// TwinCAT 3 PLC project mobject_graph_vision_pack
// Title: mobject-graph-vision-pack
// Company: mobject
// Author: mobject dev team
// ProjectVersion: 0.11.0
// ProgramVersion: 3.1.4026.25
// libraries:
//   mobject-core,0.10.0,mobject
//   mobject-graph,0.18.0,mobject
//   mobject-graph-plc-pack,0.19.0,mobject
//   Tc2_Standard, * (Beckhoff Automation GmbH)
//   Tc2_System, * (Beckhoff Automation GmbH)
//   Tc2_Utilities, * (Beckhoff Automation GmbH)
//   Tc3_Module, * (Beckhoff Automation GmbH)
//   Tc3_Vision, 5.10.2.0 (Beckhoff Automation GmbH)
// project tree:
//   Datatypes/Aliases/ _GVCP_REGISTER_ADDRESS.TcPOU, _TcVnMatrix2x3_LREAL.TcPOU, _TcVnArray4_Point2_REAL.TcPOU (not stored), _TcVnArray4_LREAL.TcPOU (not stored), _TcVnArray33_UDINT.TcPOU (not stored), _TcVnArray10_ITcVnImage.TcPOU (not stored), _TcVnArray3_Point2_REAL.TcPOU (not stored), _TcVnArray7_LREAL.TcPOU, _TcVnArray8_LREAL.TcPOU, _TcVnMatrix3x3_LREAL.TcPOU (not stored), _TcVnPoint.TcPOU (not stored), _TcVnPoint2_LREAL.TcPOU (not stored), _TcVnPoint3_REAL.TcPOU, _TcVnPoint3_LREAL.TcPOU, _TcVnPoint2_REAL.TcPOU (not stored), _TcVnRectangle.TcPOU (not stored), _TcVnVector2_DINT.TcPOU, _TcVnPoint2_DINT.TcPOU (not stored), _ALIASTYP.TcPOU (not stored) (excluded from build), _TcVnVector2_INT.TcPOU (not stored), _TcVnVector3_SINT.TcPOU (not stored), _TcVnVector3_INT.TcPOU, _TcVnVector2_SINT.TcPOU (not stored), _TcVnVector2_LREAL.TcPOU (not stored), _TcVnVector2_UINT.TcPOU (not stored), _TcVnVector2_USINT.TcPOU, _TcVnVector3_UINT.TcPOU, _TcVnVector3_USINT.TcPOU (not stored), _TcVnVector4_INT.TcPOU (not stored), _TcVnVector4_REAL.TcPOU, _TcVnVector4_SINT.TcPOU (not stored), _TcVnVector4_LREAL.TcPOU (not stored), _TcVnVector3_REAL.TcPOU, _TcVnVector3_LREAL.TcPOU (not stored), _TcVnVector2_REAL.TcPOU (not stored), _TcVnVector4_DINT.TcPOU, _TcVnVector4_UINT.TcPOU, _TcVnVector4_USINT.TcPOU, _GVCP_REGISTER_VALUE.TcPOU
//   Datatypes/Arrays/ _Array0to1OfARRAYTYP.TcPOU (not stored) (excluded from build), _Array0to1OfDINT.TcPOU (not stored), _Array0to1OfINT.TcPOU, _Array0to1OfLREAL.TcPOU (not stored), _Array0to1OfREAL.TcPOU (not stored), _Array0to1OfSINT.TcPOU, _Array0to1OfUINT.TcPOU (not stored), _Array0to1OfUSINT.TcPOU, _Array0to1_0to2OfLREAL.TcPOU, _Array0to2_0to2OfLREAL.TcPOU (not stored), _Array0to2OfINT.TcPOU (not stored), _Array0to2OfLREAL.TcPOU (not stored), _Array0to2OfREAL.TcPOU, _Array0to2OfSINT.TcPOU, _Array0to2OfTcVnPoint2_REAL.TcPOU (not stored), _Array0to2OfUINT.TcPOU (not stored), _Array0to2OfUSINT.TcPOU (not stored), _Array0to32OfUDINT.TcPOU (not stored), _Array0to3OfDINT.TcPOU (not stored), _Array0to3OfINT.TcPOU, _Array0to3OfLREAL.TcPOU, _Array0to3OfREAL.TcPOU, _Array0to3OfSINT.TcPOU (not stored), _Array0to3OfTcVnPoint2_REAL.TcPOU, _Array0to3OfUINT.TcPOU, _Array0to3OfUSINT.TcPOU (not stored), _Array0to6OfLREAL.TcPOU (not stored), _Array0to7OfLREAL.TcPOU, _Array0to9OfITcVnImage.TcPOU
//   Datatypes/Enums/ _ETcVn2dCodeSearchStrategy.TcPOU (not stored), _ETcVnCodeType.TcPOU, _ETcVnMatchTemplateWalshOptions.TcPOU, _ETcVnCodeDetectionModel.TcPOU, _ETcVnAdaptiveThresholdMethod.TcPOU (not stored), _ETcVnBarcodeSearchDirection.TcPOU (not stored), _ETcVnBarcodeType.TcPOU (not stored), _ETcVnBlobCombination.TcPOU (not stored), _ETcVnBorderInterpolationMethod.TcPOU (not stored), _ETcVnBoostClassifierType.TcPOU, _ETcVnCalibrationPattern.TcPOU (not stored), _ETcVnCalibrationPatternOrigin.TcPOU, _ETcVnCameraState.TcPOU, _ETcVnClusteringAlgorithm.TcPOU, _ETcVnColorMap.TcPOU (not stored), _ETcVnColorMapSize.TcPOU, _ETcVnColorSpaceTransform.TcPOU, _ETcVnColorTrainingMethod.TcPOU, _ETcVnConnectedComponentsAlgorithm.TcPOU, _ETcVnContainerExportFormat.TcPOU (not stored), _ETcVnContourApproximationMethod.TcPOU (not stored), _ETcVnContourRetrievalMode.TcPOU (not stored), _ETcVnContoursMatchComparisonMethod.TcPOU (not stored), _ETcVnDataMatrixOptions.TcPOU, _ETcVnFindTemplateWalshOptions.TcPOU, _ETcVnReduceType.TcPOU, _ETcVnDiffusivityTypeKAZE.TcPOU (not stored), _ETcVnDistanceTransformationLabel.TcPOU, _ETcVnDistanceTransformationMask.TcPOU, _ETcVnDistanceType.TcPOU, _ETcVnDrawMatchesFlags.TcPOU, _ETcVnDrawShape.TcPOU, _ETcVnEdgeDetectionAlgorithm.TcPOU (not stored), _ETcVnEdgeDirection.TcPOU, _ETcVnElementType.TcPOU (not stored), _ETcVnEstimationAlgorithm.TcPOU (not stored), _ETcVnExtremePointDirection.TcPOU, _ETcVnFeatureDescriptorTypeAKAZE.TcPOU, _ETcVnFeatureScalingType.TcPOU, _ETcVnFeatureScoreTypeORB.TcPOU (not stored), _ETcVnFilterDirection.TcPOU (not stored), _ETcVnFlipAxis.TcPOU, _ETcVnDataLayout.TcPOU, _ETcVnFontType.TcPOU, _ETcVnHoughMethod.TcPOU (not stored), _ETcVnInitializableFunction.TcPOU, _ETcVnInterpolationType.TcPOU (not stored), _ETcVnKeypointDetectionTypeAGAST.TcPOU, _ETcVnKeypointDetectionTypeFAST.TcPOU (not stored), _ETcVnKnn.TcPOU (not stored), _ETcVnLineType.TcPOU, _ETcVnMorphologicalOperator.TcPOU, _ETcVnNbc.TcPOU (not stored), _ETcVnNormalizationType.TcPOU (not stored), _ETcVnOcrModelType.TcPOU, _ETcVnCircularityCalculationMethod.TcPOU, _ETcVnLayerNameType.TcPOU, _ETcVnTimestamp.TcPOU, _ETcVnOcrOptions.TcPOU, _ETcVnOrientationMethod.TcPOU (not stored), _ETcVnPaddingMode.TcPOU (not stored), _ETcVnPixelConnectivity.TcPOU, _ETcVnPixelEncoding.TcPOU (not stored), _ETcVnPixelPackMode.TcPOU, _ETcVnPrototypeClusterer.TcPOU (not stored), _ETcVnRectangleIntersection.TcPOU, _ETcVnRotationAngle.TcPOU, _ETcVnRTrees.TcPOU (not stored), _ETcVnSignedNormalization.TcPOU (not stored), _ETcVnSolvePnPMethod.TcPOU (not stored), _ETcVnSta.TcPOU (not stored), _ETcVnStructuringElementShape.TcPOU, _ETcVnSvm.TcPOU (not stored), _ETcVnSvmKernelType.TcPOU (not stored), _ETcVnSvmSgdClassifierMarginType.TcPOU, _ETcVnSvmSgdClassifierType.TcPOU (not stored), _ETcVnTemplateMatchMethod.TcPOU (not stored), _ETcVnThresholdType.TcPOU, _ETcVnVectorCompareMethod.TcPOU (not stored), _ETcVnWorldCoordinateSystem.TcPOU (not stored), _ETcWatchdogAccumulationType.TcPOU (not stored), _GEV_CAMERA_STATE.TcPOU, _ETcVnComparisonOperator.TcPOU, _ETcVnDetectBarcodesWalshOptions.TcPOU, _ETcVnDetectPatternPointsOptions.TcPOU, _ETcVnDotCodeOptions.TcPOU, _ETcVnEdgeSelection.TcPOU, _ETcVnFindRoisMethod.TcPOU, _ETcVnJpegSampling.TcPOU, _ETcVnMergeRegionsOptions.TcPOU, _ETcVnPolarizedImageInterpolation.TcPOU, _ETcVnSalientFeaturesMethod.TcPOU
//   Datatypes/Interfaces/Containers/ITcVnContainer/ I_InterfaceDatatype_ITcVnContainer.TcIO (not stored), _ITcVnContainer.TcPOU (not stored)
//   Datatypes/Interfaces/Containers/Iterators/ITcVnBidirectionalIterator/ I_InterfaceDatatype_ITcVnBidirectionalIterator.TcIO (not stored), _ITcVnBidirectionalIterator.TcPOU (not stored)
//   Datatypes/Interfaces/Images/ITcVnImage/ I_InterfaceDatatype_ITcVnImage.TcIO (not stored), _ITcVnImage.TcPOU (not stored)
//   Datatypes/Interfaces/Images/ITcVnDisplayableImage/ I_InterfaceDatatype_ITcVnDisplayableImage.TcIO (not stored), _ITcVnDisplayableImage.TcPOU (not stored)
//   Datatypes/Structs/ _GVSP_LEADER_PAYLOAD_IMAGE.TcPOU, _GVSP_IMAGE_INFO.TcPOU, _TcVnCodeGradesDM.TcPOU, _TcVnCodeGradesQR.TcPOU, _TcVnMoments.TcPOU, _TcVnDMatch.TcPOU, _GVSP_PIXEL_FORMAT.TcPOU, _TcVnKeyPoint.TcPOU (not stored), _TcVnImageInfo.TcPOU (not stored), _TcVnCodeGrades1D.TcPOU, _TcVnMatrix.TcPOU (excluded from build), _TcVnParamsMSER.TcPOU, _TcVnParamsKAZE.TcPOU (not stored), _TcVnParamsAKAZE.TcPOU, _TcVnParamsORB.TcPOU (not stored), _TcVnParamsSB.TcPOU, _TcVnParamsBRISK.TcPOU, _TcVnParamsFAST.TcPOU, _TcVnParamsBlobDetection.TcPOU, _TcVnParamsAGAST.TcPOU (not stored), _TcVnCameraCalibrationOptions.TcPOU, _TcVnParamsGFTT.TcPOU, _TcVnRotatedRectangle.TcPOU, _TcVnCircularArc.TcPOU, _TcVnSize2_REAL.TcPOU (not stored), _TcVnPixelFormat.TcPOU, _TcVnRectangle_DINT.TcPOU, _TcVnRectangle_UDINT.TcPOU, _GVCP_ADDRESS_VALUE_PAIR.TcPOU, _TcVnSize2_DINT.TcPOU, _TcVnParamsFindRois.TcPOU, _TcVnParamsWalshBarcodeDetection.TcPOU
//   Datatypes/ VisionDatatypePack.TcPOU
//   Extensions/PreExecutionCheck/Alarms/ PreExecutionCheckFailedAlarm.TcPOU (not stored)
//   Extensions/PreExecutionCheck/Checks/ I_PreExecutionChecks.TcIO (not stored), PreExecutionChecks.TcPOU (not stored)
//   Extensions/PreExecutionCheck/Interfaces/ I_PreCheckedNode.TcIO (not stored)
//   Extensions/PreExecutionCheck/ PreExecutionCheckExtension.TcPOU
//   Extensions/WatchdogCheck/ WatchdogCheckExtension.TcPOU
//   Functions/Checks/ ContainersHaveMatchingNumberOfElements.TcPOU, ImageHasCompatibleElementType.TcPOU, ImageHasElementType.TcPOU, ImagesHaveMatchingChannels.TcPOU, ContainersHaveMatchingTypes.TcPOU, ImagesHaveMatchingPixelFormats.TcPOU, IsImage1SizeEqualToImage2Size.TcPOU, IsImage1WidthEqualToImage2Width.TcPOU, IsMaxValueCompatibleWithPixelDepth.TcPOU, IsTemplateImageSmallerThanSourceImage.TcPOU, IsRoiSizeOK_Udint.TcPOU, IsRoiSizeOK_Dint.TcPOU, IsValidImage.TcPOU, IsValidContainer.TcPOU, IsValidIterator.TcPOU, IsRemapMapPairValid.TcPOU
//   Functions/Helpers/ GetETcVnElementTypeFromImage.TcPOU
//   / GVL_COLOURS.TcGVL, VisionPack.TcPOU
//   Nodes/Algebraic Container Ops/AddTo/ Node_F_VN_AddToContainerElements_DINT.TcPOU (not stored), Node_F_VN_AddToContainerElements_INT.TcPOU (not stored), Node_F_VN_AddToContainerElements_LREAL.TcPOU (not stored), Node_F_VN_AddToContainerElements_REAL.TcPOU (not stored), Node_F_VN_AddToContainerElements_SINT.TcPOU (not stored), Node_F_VN_AddToContainerElements_TcVnKeyPoint.TcPOU (not stored), Node_F_VN_AddToContainerElements_TcVnPoint2_DINT.TcPOU (not stored), Node_F_VN_AddToContainerElements_TcVnPoint2_LREAL.TcPOU (not stored), Node_F_VN_AddToContainerElements_TcVnPoint2_REAL.TcPOU (not stored), Node_F_VN_AddToContainerElements_TcVnPoint3_LREAL.TcPOU (not stored), Node_F_VN_AddToContainerElements_TcVnPoint3_REAL.TcPOU (not stored), Node_F_VN_AddToContainerElements_TcVnRectangle_DINT.TcPOU (not stored), Node_F_VN_AddToContainerElements_TcVnRotatedRectangle.TcPOU (not stored), Node_F_VN_AddToContainerElements_TcVnVector2_DINT.TcPOU (not stored), Node_F_VN_AddToContainerElements_TcVnVector2_INT.TcPOU (not stored), Node_F_VN_AddToContainerElements_TcVnVector2_REAL.TcPOU (not stored), Node_F_VN_AddToContainerElements_TcVnVector2_SINT.TcPOU (not stored), Node_F_VN_AddToContainerElements_TcVnVector2_UINT.TcPOU (not stored), Node_F_VN_AddToContainerElements_TcVnVector2_USINT.TcPOU (not stored), Node_F_VN_AddToContainerElements_TcVnVector3_INT.TcPOU (not stored), Node_F_VN_AddToContainerElements_TcVnVector3_REAL.TcPOU (not stored), Node_F_VN_AddToContainerElements_TcVnVector3_SINT.TcPOU (not stored), Node_F_VN_AddToContainerElements_TcVnVector3_UINT.TcPOU (not stored), Node_F_VN_AddToContainerElements_TcVnVector3_USINT.TcPOU (not stored), Node_F_VN_AddToContainerElements_TcVnVector4_DINT.TcPOU (not stored), Node_F_VN_AddToContainerElements_TcVnVector4_INT.TcPOU (not stored), Node_F_VN_AddToContainerElements_TcVnVector4_LREAL.TcPOU (not stored), Node_F_VN_AddToContainerElements_TcVnVector4_REAL.TcPOU (not stored), Node_F_VN_AddToContainerElements_TcVnVector4_SINT.TcPOU (not stored), Node_F_VN_AddToContainerElements_TcVnVector4_UINT.TcPOU (not stored), Node_F_VN_AddToContainerElements_TcVnVector4_USINT.TcPOU (not stored), Node_F_VN_AddToContainerElements_UDINT.TcPOU (not stored), Node_F_VN_AddToContainerElements_UINT.TcPOU (not stored), Node_F_VN_AddToContainerElements_ULINT.TcPOU (not stored), Node_F_VN_AddToContainerElements_USINT.TcPOU (not stored)
//   Nodes/Algebraic Container Ops/ Node_F_VN_AddContainers.TcPOU, Node_F_VN_BitwiseNotContainer.TcPOU, Node_F_VN_BitwiseOrContainers.TcPOU, Node_F_VN_BitwiseXorContainers.TcPOU, Node_F_VN_DivideContainersExp.TcPOU, Node_F_VN_BitwiseAndContainers.TcPOU, Node_F_VN_MaxContainer.TcPOU, Node_F_VN_MinContainer.TcPOU, Node_F_VN_MultiplyContainers.TcPOU, Node_F_VN_DivideContainers.TcPOU, Node_F_VN_NegateContainer.TcPOU, Node_F_VN_SubtractContainers.TcPOU
//   Nodes/Algebraic Image Ops/ Node_F_VN_AddImages.TcPOU, Node_F_VN_AddImagesWeighted.TcPOU, Node_F_VN_AddImagesWeightedExp.TcPOU, Node_F_VN_AddVectorToImage.TcPOU, Node_F_VN_BitwiseAndImagesExp.TcPOU, Node_F_VN_BitwiseNotImageExp.TcPOU, Node_F_VN_MaxImageExp.TcPOU, Node_F_VN_BitwiseXorImagesExp.TcPOU, Node_F_VN_BitwiseOrImagesExp.TcPOU, Node_F_VN_BitwiseAndScalarWithImage.TcPOU, Node_F_VN_BitwiseXorVectorWithImage.TcPOU, Node_F_VN_BitwiseXorScalarWithImage.TcPOU, Node_F_VN_BitwiseOrVectorWithImage.TcPOU, Node_F_VN_BitwiseOrScalarWithImage.TcPOU, Node_F_VN_BitwiseAndVectorWithImage.TcPOU, Node_F_VN_DivideImageByScalar.TcPOU, Node_F_VN_DivideVectorByImage.TcPOU, Node_F_VN_DivideScalarByImage.TcPOU, Node_F_VN_DivideImageByVector.TcPOU, Node_F_VN_ElementwiseExp.TcPOU, Node_F_VN_ElementwiseLog.TcPOU, Node_F_VN_MaxImageWithScalarExp.TcPOU, Node_F_VN_MaxImageWithVectorExp.TcPOU, Node_F_VN_MinImageWithVectorExp.TcPOU, Node_F_VN_MinImageWithScalarExp.TcPOU, Node_F_VN_MinImageExp.TcPOU, Node_F_VN_MaxImageWithScalar.TcPOU, Node_F_VN_MinImageWithVector.TcPOU, Node_F_VN_MinImageWithScalar.TcPOU, Node_F_VN_MaxImageWithVector.TcPOU, Node_F_VN_MultiplyImageWithScalar.TcPOU, Node_F_VN_MultiplyImageWithVector.TcPOU, Node_F_VN_SubtractImageFromVector.TcPOU, Node_F_VN_SubtractScalarFromImage.TcPOU, Node_F_VN_MultiplyImages.TcPOU, Node_F_VN_SubtractImages.TcPOU, Node_F_VN_MaxImage.TcPOU, Node_F_VN_BitwiseOrImages.TcPOU, Node_F_VN_BitwiseNotImage.TcPOU, Node_F_VN_BitwiseAndImages.TcPOU, Node_F_VN_BitwiseXorImages.TcPOU, Node_F_VN_MinImage.TcPOU, Node_F_VN_DivideImages.TcPOU, Node_F_VN_SubtractImageFromScalar.TcPOU, Node_F_VN_AddScalarToImage.TcPOU, Node_F_VN_SubtractVectorFromImage.TcPOU
//   Nodes/Basic Container Ops/AppendToContainer/ Node_F_VN_AppendToContainer_DINT.TcPOU (not stored), Node_F_VN_AppendToContainer_INT.TcPOU (not stored), Node_F_VN_AppendToContainer_ITcVnContainer.TcPOU (not stored), Node_F_VN_AppendToContainer_ITcVnImage.TcPOU (not stored), Node_F_VN_AppendToContainer_LREAL.TcPOU (not stored), Node_F_VN_AppendToContainer_REAL.TcPOU (not stored), Node_F_VN_AppendToContainer_SINT.TcPOU (not stored), Node_F_VN_AppendToContainer_TcVnDMatch.TcPOU (not stored), Node_F_VN_AppendToContainer_TcVnKeyPoint.TcPOU (not stored), Node_F_VN_AppendToContainer_TcVnPoint2_DINT.TcPOU (not stored), Node_F_VN_AppendToContainer_TcVnPoint2_LREAL.TcPOU (not stored), Node_F_VN_AppendToContainer_TcVnPoint2_REAL.TcPOU (not stored), Node_F_VN_AppendToContainer_TcVnPoint3_LREAL.TcPOU (not stored), Node_F_VN_AppendToContainer_TcVnPoint3_REAL.TcPOU (not stored), Node_F_VN_AppendToContainer_TcVnRectangle_DINT.TcPOU (not stored), Node_F_VN_AppendToContainer_TcVnRotatedRectangle.TcPOU (not stored), Node_F_VN_AppendToContainer_TcVnVector2_DINT.TcPOU (not stored), Node_F_VN_AppendToContainer_TcVnVector2_INT.TcPOU (not stored), Node_F_VN_AppendToContainer_TcVnVector2_REAL.TcPOU (not stored), Node_F_VN_AppendToContainer_TcVnVector2_SINT.TcPOU (not stored), Node_F_VN_AppendToContainer_TcVnVector2_UINT.TcPOU (not stored), Node_F_VN_AppendToContainer_TcVnVector2_USINT.TcPOU (not stored), Node_F_VN_AppendToContainer_TcVnVector3_INT.TcPOU (not stored), Node_F_VN_AppendToContainer_TcVnVector3_REAL.TcPOU (not stored), Node_F_VN_AppendToContainer_TcVnVector3_SINT.TcPOU (not stored), Node_F_VN_AppendToContainer_TcVnVector3_UINT.TcPOU (not stored), Node_F_VN_AppendToContainer_TcVnVector3_USINT.TcPOU (not stored), Node_F_VN_AppendToContainer_TcVnVector4_DINT.TcPOU (not stored), Node_F_VN_AppendToContainer_TcVnVector4_INT.TcPOU (not stored), Node_F_VN_AppendToContainer_TcVnVector4_LREAL.TcPOU (not stored), Node_F_VN_AppendToContainer_TcVnVector4_REAL.TcPOU (not stored), Node_F_VN_AppendToContainer_TcVnVector4_SINT.TcPOU (not stored), Node_F_VN_AppendToContainer_TcVnVector4_UINT.TcPOU (not stored), Node_F_VN_AppendToContainer_TcVnVector4_USINT.TcPOU (not stored), Node_F_VN_AppendToContainer_UDINT.TcPOU (not stored), Node_F_VN_AppendToContainer_UINT.TcPOU (not stored), Node_F_VN_AppendToContainer_ULINT.TcPOU (not stored), Node_F_VN_AppendToContainer_USINT.TcPOU (not stored), Node_F_VN_FillContainer_TcVnVector4_REAL.TcPOU (not stored)
//   Nodes/Basic Container Ops/FillContainerExp/ Node_F_VN_FillContainerExp_DINT.TcPOU (not stored), Node_F_VN_FillContainerExp_INT.TcPOU (not stored), Node_F_VN_FillContainerExp_ITcVnImage.TcPOU (not stored), Node_F_VN_FillContainerExp_LREAL.TcPOU (not stored), Node_F_VN_FillContainerExp_REAL.TcPOU (not stored), Node_F_VN_FillContainerExp_SINT.TcPOU (not stored), Node_F_VN_FillContainerExp_TcVnDMatch.TcPOU (not stored), Node_F_VN_FillContainerExp_TcVnKeyPoint.TcPOU (not stored), Node_F_VN_FillContainerExp_TcVnPoint2_DINT.TcPOU (not stored), Node_F_VN_FillContainerExp_TcVnPoint2_LREAL.TcPOU (not stored), Node_F_VN_FillContainerExp_TcVnPoint2_REAL.TcPOU (not stored), Node_F_VN_FillContainerExp_TcVnPoint3_LREAL.TcPOU (not stored), Node_F_VN_FillContainerExp_TcVnPoint3_REAL.TcPOU (not stored), Node_F_VN_FillContainerExp_TcVnRectangle_DINT.TcPOU (not stored), Node_F_VN_FillContainerExp_TcVnRotatedRectangle.TcPOU (not stored), Node_F_VN_FillContainerExp_TcVnVector2_DINT.TcPOU (not stored), Node_F_VN_FillContainerExp_TcVnVector2_INT.TcPOU (not stored), Node_F_VN_FillContainerExp_TcVnVector2_REAL.TcPOU (not stored), Node_F_VN_FillContainerExp_TcVnVector2_SINT.TcPOU (not stored), Node_F_VN_FillContainerExp_TcVnVector2_UINT.TcPOU (not stored), Node_F_VN_FillContainerExp_TcVnVector2_USINT.TcPOU (not stored), Node_F_VN_FillContainerExp_TcVnVector3_INT.TcPOU (not stored), Node_F_VN_FillContainerExp_TcVnVector3_REAL.TcPOU (not stored), Node_F_VN_FillContainerExp_TcVnVector3_SINT.TcPOU (not stored), Node_F_VN_FillContainerExp_TcVnVector3_UINT.TcPOU (not stored), Node_F_VN_FillContainerExp_TcVnVector3_USINT.TcPOU (not stored), Node_F_VN_FillContainerExp_TcVnVector4_DINT.TcPOU (not stored), Node_F_VN_FillContainerExp_TcVnVector4_INT.TcPOU (not stored), Node_F_VN_FillContainerExp_TcVnVector4_LREAL.TcPOU (not stored), Node_F_VN_FillContainerExp_TcVnVector4_REAL.TcPOU (not stored), Node_F_VN_FillContainerExp_TcVnVector4_SINT.TcPOU (not stored), Node_F_VN_FillContainerExp_TcVnVector4_UINT.TcPOU (not stored), Node_F_VN_FillContainerExp_TcVnVector4_USINT.TcPOU (not stored), Node_F_VN_FillContainerExp_UDINT.TcPOU (not stored), Node_F_VN_FillContainerExp_UINT.TcPOU (not stored), Node_F_VN_FillContainerExp_ULINT.TcPOU (not stored), Node_F_VN_FillContainerExp_USINT.TcPOU (not stored)
//   Nodes/Basic Container Ops/FillContainer/ Node_F_VN_FillContainer_DINT.TcPOU (not stored), Node_F_VN_FillContainer_INT.TcPOU (not stored), Node_F_VN_FillContainer_ITcVnImage.TcPOU (not stored), Node_F_VN_FillContainer_LREAL.TcPOU (not stored), Node_F_VN_FillContainer_REAL.TcPOU (not stored), Node_F_VN_FillContainer_SINT.TcPOU (not stored), Node_F_VN_FillContainer_TcVnDMatch.TcPOU (not stored), Node_F_VN_FillContainer_TcVnKeyPoint.TcPOU (not stored), Node_F_VN_FillContainer_TcVnPoint2_DINT.TcPOU (not stored), Node_F_VN_FillContainer_TcVnPoint2_LREAL.TcPOU (not stored), Node_F_VN_FillContainer_TcVnPoint2_REAL.TcPOU (not stored), Node_F_VN_FillContainer_TcVnPoint3_LREAL.TcPOU (not stored), Node_F_VN_FillContainer_TcVnPoint3_REAL.TcPOU (not stored), Node_F_VN_FillContainer_TcVnRectangle_DINT.TcPOU (not stored), Node_F_VN_FillContainer_TcVnRotatedRectangle.TcPOU (not stored), Node_F_VN_FillContainer_TcVnVector2_DINT.TcPOU (not stored), Node_F_VN_FillContainer_TcVnVector2_INT.TcPOU (not stored), Node_F_VN_FillContainer_TcVnVector2_REAL.TcPOU (not stored), Node_F_VN_FillContainer_TcVnVector2_SINT.TcPOU (not stored), Node_F_VN_FillContainer_TcVnVector2_UINT.TcPOU (not stored), Node_F_VN_FillContainer_TcVnVector2_USINT.TcPOU (not stored), Node_F_VN_FillContainer_TcVnVector3_INT.TcPOU (not stored), Node_F_VN_FillContainer_TcVnVector3_REAL.TcPOU (not stored), Node_F_VN_FillContainer_TcVnVector3_SINT.TcPOU (not stored), Node_F_VN_FillContainer_TcVnVector3_UINT.TcPOU (not stored), Node_F_VN_FillContainer_TcVnVector3_USINT.TcPOU (not stored), Node_F_VN_FillContainer_TcVnVector4_DINT.TcPOU (not stored), Node_F_VN_FillContainer_TcVnVector4_INT.TcPOU (not stored), Node_F_VN_FillContainer_TcVnVector4_LREAL.TcPOU (not stored), Node_F_VN_FillContainer_TcVnVector4_SINT.TcPOU (not stored), Node_F_VN_FillContainer_TcVnVector4_UINT.TcPOU (not stored), Node_F_VN_FillContainer_TcVnVector4_USINT.TcPOU (not stored), Node_F_VN_FillContainer_UDINT.TcPOU (not stored), Node_F_VN_FillContainer_UINT.TcPOU (not stored), Node_F_VN_FillContainer_ULINT.TcPOU (not stored), Node_F_VN_FillContainer_USINT.TcPOU (not stored)
//   Nodes/Basic Container Ops/GetAt/ Node_F_VN_GetAt_DINT.TcPOU (not stored), Node_F_VN_GetAt_INT.TcPOU (not stored), Node_F_VN_GetAt_ITcVnContainer.TcPOU (not stored), Node_F_VN_GetAt_ITcVnImage.TcPOU (not stored), Node_F_VN_GetAt_LREAL.TcPOU (not stored), Node_F_VN_GetAt_REAL.TcPOU (not stored), Node_F_VN_GetAt_SINT.TcPOU (not stored), Node_F_VN_GetAt_TcVnDMatch.TcPOU (not stored), Node_F_VN_GetAt_TcVnKeyPoint.TcPOU (not stored), Node_F_VN_GetAt_TcVnPoint2_DINT.TcPOU (not stored), Node_F_VN_GetAt_TcVnPoint2_LREAL.TcPOU (not stored), Node_F_VN_GetAt_TcVnPoint2_REAL.TcPOU (not stored), Node_F_VN_GetAt_TcVnPoint3_LREAL.TcPOU (not stored), Node_F_VN_GetAt_TcVnPoint3_REAL.TcPOU (not stored), Node_F_VN_GetAt_TcVnRectangle_DINT.TcPOU (not stored), Node_F_VN_GetAt_TcVnRotatedRectangle.TcPOU (not stored), Node_F_VN_GetAt_TcVnVector2_DINT.TcPOU (not stored), Node_F_VN_GetAt_TcVnVector2_INT.TcPOU (not stored), Node_F_VN_GetAt_TcVnVector2_REAL.TcPOU (not stored), Node_F_VN_GetAt_TcVnVector2_SINT.TcPOU (not stored), Node_F_VN_GetAt_TcVnVector2_UINT.TcPOU (not stored), Node_F_VN_GetAt_TcVnVector2_USINT.TcPOU (not stored), Node_F_VN_GetAt_TcVnVector3_INT.TcPOU (not stored), Node_F_VN_GetAt_TcVnVector3_REAL.TcPOU (not stored), Node_F_VN_GetAt_TcVnVector3_SINT.TcPOU (not stored), Node_F_VN_GetAt_TcVnVector3_UINT.TcPOU (not stored), Node_F_VN_GetAt_TcVnVector3_USINT.TcPOU (not stored), Node_F_VN_GetAt_TcVnVector4_DINT.TcPOU (not stored), Node_F_VN_GetAt_TcVnVector4_INT.TcPOU (not stored), Node_F_VN_GetAt_TcVnVector4_LREAL.TcPOU (not stored), Node_F_VN_GetAt_TcVnVector4_REAL.TcPOU (not stored), Node_F_VN_GetAt_TcVnVector4_SINT.TcPOU (not stored), Node_F_VN_GetAt_TcVnVector4_UINT.TcPOU (not stored), Node_F_VN_GetAt_TcVnVector4_USINT.TcPOU (not stored), Node_F_VN_GetAt_UDINT.TcPOU (not stored), Node_F_VN_GetAt_UINT.TcPOU (not stored), Node_F_VN_GetAt_ULINT.TcPOU (not stored), Node_F_VN_GetAt_USINT.TcPOU (not stored)
//   Nodes/Basic Container Ops/InsertIntoContainer/ Node_F_VN_InsertIntoContainer_DINT.TcPOU (not stored), Node_F_VN_InsertIntoContainer_INT.TcPOU (not stored), Node_F_VN_InsertIntoContainer_ITcVnContainer.TcPOU (not stored), Node_F_VN_InsertIntoContainer_ITcVnImage.TcPOU (not stored), Node_F_VN_InsertIntoContainer_LREAL.TcPOU (not stored), Node_F_VN_InsertIntoContainer_REAL.TcPOU (not stored), Node_F_VN_InsertIntoContainer_SINT.TcPOU (not stored), Node_F_VN_InsertIntoContainer_TcVnDMatch.TcPOU (not stored), Node_F_VN_InsertIntoContainer_TcVnKeyPoint.TcPOU (not stored), Node_F_VN_InsertIntoContainer_TcVnPoint2_DINT.TcPOU (not stored), Node_F_VN_InsertIntoContainer_TcVnPoint2_LREAL.TcPOU (not stored), Node_F_VN_InsertIntoContainer_TcVnPoint2_REAL.TcPOU (not stored), Node_F_VN_InsertIntoContainer_TcVnPoint3_LREAL.TcPOU (not stored), Node_F_VN_InsertIntoContainer_TcVnPoint3_REAL.TcPOU (not stored), Node_F_VN_InsertIntoContainer_TcVnRectangle_DINT.TcPOU (not stored), Node_F_VN_InsertIntoContainer_TcVnRotatedRectangle.TcPOU (not stored), Node_F_VN_InsertIntoContainer_TcVnVector2_DINT.TcPOU (not stored), Node_F_VN_InsertIntoContainer_TcVnVector2_INT.TcPOU (not stored), Node_F_VN_InsertIntoContainer_TcVnVector2_REAL.TcPOU (not stored), Node_F_VN_InsertIntoContainer_TcVnVector2_SINT.TcPOU (not stored), Node_F_VN_InsertIntoContainer_TcVnVector2_UINT.TcPOU (not stored), Node_F_VN_InsertIntoContainer_TcVnVector2_USINT.TcPOU (not stored), Node_F_VN_InsertIntoContainer_TcVnVector3_INT.TcPOU (not stored), Node_F_VN_InsertIntoContainer_TcVnVector3_REAL.TcPOU (not stored), Node_F_VN_InsertIntoContainer_TcVnVector3_SINT.TcPOU (not stored), Node_F_VN_InsertIntoContainer_TcVnVector3_UINT.TcPOU (not stored), Node_F_VN_InsertIntoContainer_TcVnVector3_USINT.TcPOU (not stored), Node_F_VN_InsertIntoContainer_TcVnVector4_DINT.TcPOU (not stored), Node_F_VN_InsertIntoContainer_TcVnVector4_INT.TcPOU (not stored), Node_F_VN_InsertIntoContainer_TcVnVector4_LREAL.TcPOU (not stored), Node_F_VN_InsertIntoContainer_TcVnVector4_REAL.TcPOU (not stored), Node_F_VN_InsertIntoContainer_TcVnVector4_SINT.TcPOU (not stored), Node_F_VN_InsertIntoContainer_TcVnVector4_UINT.TcPOU (not stored), Node_F_VN_InsertIntoContainer_TcVnVector4_USINT.TcPOU (not stored), Node_F_VN_InsertIntoContainer_UDINT.TcPOU (not stored), Node_F_VN_InsertIntoContainer_UINT.TcPOU (not stored), Node_F_VN_InsertIntoContainer_ULINT.TcPOU (not stored), Node_F_VN_InsertIntoContainer_USINT.TcPOU (not stored)
//   Nodes/Basic Container Ops/ Node_F_VN_CreateContainer.TcPOU, Node_F_VN_ExportContainer_String.TcPOU, Node_F_VN_ExtractContainerRange.TcPOU, Node_F_VN_ReverseContainer.TcPOU, Node_F_VN_GetNumberOfElements.TcPOU, Node_F_VN_ExportSubContainer_String.TcPOU, Node_F_VN_CheckIfEmpty.TcPOU, Node_F_VN_CopyContainer.TcPOU
//   Nodes/Basic Container Ops/SetAt/ Node_F_VN_SetAt_DINT.TcPOU (not stored), Node_F_VN_SetAt_INT.TcPOU (not stored), Node_F_VN_SetAt_ITcVnContainer.TcPOU (not stored), Node_F_VN_SetAt_ITcVnImage.TcPOU (not stored), Node_F_VN_SetAt_LREAL.TcPOU (not stored), Node_F_VN_SetAt_REAL.TcPOU (not stored), Node_F_VN_SetAt_SINT.TcPOU (not stored), Node_F_VN_SetAt_TcVnDMatch.TcPOU (not stored), Node_F_VN_SetAt_TcVnKeyPoint.TcPOU (not stored), Node_F_VN_SetAt_TcVnPoint2_DINT.TcPOU (not stored), Node_F_VN_SetAt_TcVnPoint2_LREAL.TcPOU (not stored), Node_F_VN_SetAt_TcVnPoint2_REAL.TcPOU (not stored), Node_F_VN_SetAt_TcVnPoint3_LREAL.TcPOU (not stored), Node_F_VN_SetAt_TcVnPoint3_REAL.TcPOU (not stored), Node_F_VN_SetAt_TcVnRectangle_DINT.TcPOU (not stored), Node_F_VN_SetAt_TcVnRotatedRectangle.TcPOU (not stored), Node_F_VN_SetAt_TcVnVector2_DINT.TcPOU (not stored), Node_F_VN_SetAt_TcVnVector2_INT.TcPOU (not stored), Node_F_VN_SetAt_TcVnVector2_REAL.TcPOU (not stored), Node_F_VN_SetAt_TcVnVector2_SINT.TcPOU (not stored), Node_F_VN_SetAt_TcVnVector2_UINT.TcPOU (not stored), Node_F_VN_SetAt_TcVnVector2_USINT.TcPOU (not stored), Node_F_VN_SetAt_TcVnVector3_INT.TcPOU (not stored), Node_F_VN_SetAt_TcVnVector3_REAL.TcPOU (not stored), Node_F_VN_SetAt_TcVnVector3_SINT.TcPOU (not stored), Node_F_VN_SetAt_TcVnVector3_UINT.TcPOU (not stored), Node_F_VN_SetAt_TcVnVector3_USINT.TcPOU (not stored), Node_F_VN_SetAt_TcVnVector4_DINT.TcPOU (not stored), Node_F_VN_SetAt_TcVnVector4_INT.TcPOU (not stored), Node_F_VN_SetAt_TcVnVector4_LREAL.TcPOU (not stored), Node_F_VN_SetAt_TcVnVector4_REAL.TcPOU (not stored), Node_F_VN_SetAt_TcVnVector4_SINT.TcPOU (not stored), Node_F_VN_SetAt_TcVnVector4_UINT.TcPOU (not stored), Node_F_VN_SetAt_TcVnVector4_USINT.TcPOU (not stored), Node_F_VN_SetAt_UDINT.TcPOU (not stored), Node_F_VN_SetAt_UINT.TcPOU (not stored), Node_F_VN_SetAt_ULINT.TcPOU (not stored), Node_F_VN_SetAt_USINT.TcPOU (not stored)
//   Nodes/Basic Image Ops/ Node_F_VN_CreateNDimensionalImage.TcPOU, Node_F_VN_CreateNDimensionalImageAndSetPixels.TcPOU, Node_F_VN_ExportImageAsBmpSizeExp.TcPOU, Node_F_VN_FuseImages.TcPOU, Node_F_VN_CopyImageRegion.TcPOU, Node_F_VN_CopyImageRegionToRegion.TcPOU, Node_F_VN_ExportImageSize.TcPOU, Node_F_VN_ExportImageAsBmpSize.TcPOU, Node_F_VN_MixImageChannels.TcPOU, Node_F_VN_GetLayoutInfo.TcPOU, Node_F_VN_PadImageBorder.TcPOU, Node_F_VN_PadImageBorderExp.TcPOU, Node_F_VN_SetImageChannel.TcPOU, Node_F_VN_SetPixelsExp.TcPOU, Node_F_VN_TransformIntoDisplayableImage.TcPOU, Node_F_VN_ConvertElementType.TcPOU, Node_F_VN_ConvertElementTypeExp.TcPOU, Node_F_VN_CopyImage.TcPOU, Node_F_VN_CreateImage.TcPOU, Node_F_VN_CreateImageAndSetPixels.TcPOU, Node_F_VN_CreateEmptyImage.TcPOU, Node_F_VN_GetPixelFormat.TcPOU, Node_F_VN_ResetRoi.TcPOU, Node_F_VN_SetPixels.TcPOU, Node_F_VN_GetPixel.TcPOU, Node_F_VN_SetRoi.TcPOU, Node_F_VN_GetImageChannel.TcPOU, Node_F_VN_GetImageHeight.TcPOU, Node_F_VN_GetImageWidth.TcPOU, Node_F_VN_GetImageInfo.TcPOU, Node_F_VN_GetRoi.TcPOU, Node_F_VN_SetPixel.TcPOU, Node_F_VN_SetRoi_TcVnRectangle_DINT.TcPOU, Node_F_VN_SetRoi_TcVnRectangle_UDINT.TcPOU, Node_F_VN_TransformIntoDisplayableImageExp.TcPOU, Node_F_VN_CopyIntoDisplayableImage.TcPOU, Node_F_VN_CreateAssociatedImage.TcPOU
//   Nodes/Code Quality/ Node_F_VN_GradeBarcode.TcPOU, Node_F_VN_GradeBarcodeExp.TcPOU, Node_F_VN_GradeDataMatrixCodeExp.TcPOU, Node_F_VN_GradeQRCode.TcPOU, Node_F_VN_GradeDataMatrixCode.TcPOU, Node_F_VN_GradeQRCodeExp.TcPOU
//   Nodes/Code Reading/ Node_F_VN_DetectCodesNeuralNetwork.TcPOU, Node_F_VN_ReadBarcodeExp.TcPOU, Node_F_VN_ReadBarcodeExp2.TcPOU, Node_F_VN_ReadDataMatrixCodeExp2.TcPOU, Node_F_VN_ReadDataMatrixCodeRoi.TcPOU, Node_F_VN_AnalyzeBarcodeWalsh.TcPOU, Node_F_VN_DetectBarcodesWalsh.TcPOU, Node_F_VN_ReadBarcodeRoi.TcPOU, Node_F_VN_ReadBarcodeRoiExp.TcPOU, Node_F_VN_ReadDataMatrixCodeRoiExp.TcPOU, Node_F_VN_ReadDataMatrixCodeExp.TcPOU, Node_F_VN_ReadDotCodeRoiExp.TcPOU, Node_F_VN_ReadPharmaCodeExp.TcPOU, Node_F_VN_ReadPharmaCodeExp2.TcPOU, Node_F_VN_ReadQRCode.TcPOU, Node_F_VN_ReadDataMatrixCode.TcPOU, Node_F_VN_ReadBarcode.TcPOU, Node_F_VN_ReadPharmaCode.TcPOU, Node_F_VN_ReadQRCodeExp.TcPOU, Node_F_VN_ReadQRCodeExp2.TcPOU, Node_F_VN_ReadDotCodeRoi.TcPOU
//   Nodes/Constants/ Node_ContainerType_String_SINT.TcPOU, Node_ContainerType_Vector_UINT.TcPOU, Node_ContainerType_Vector_String_SINT.TcPOU, Node_ContainerType_Vector_Vector_TcVnDMatch.TcPOU, Node_ContainerType_Vector_TcVnDMatch.TcPOU, Node_ContainerType_Vector_TcVnKeyPoint.TcPOU, Node_ContainerType_Vector_TcVnRotatedRectangle.TcPOU, Node_ContainerType_Vector_TcVnRectangle_DINT.TcPOU, Node_ContainerType_Vector_TcVnVector4_LREAL.TcPOU, Node_ContainerType_Vector_TcVnVector4_REAL.TcPOU, Node_ContainerType_Vector_TcVnVector4_DINT.TcPOU, Node_ContainerType_Vector_TcVnVector4_UINT.TcPOU, Node_ContainerType_Vector_TcVnVector4_INT.TcPOU, Node_ContainerType_Vector_TcVnVector4_USINT.TcPOU, Node_ContainerType_Vector_TcVnVector4_SINT.TcPOU, Node_ContainerType_Vector_TcVnVector3_REAL.TcPOU, Node_ContainerType_Vector_TcVnVector3_UINT.TcPOU, Node_ContainerType_Vector_TcVnVector3_INT.TcPOU, Node_ContainerType_Vector_TcVnVector3_USINT.TcPOU, Node_ContainerType_Vector_TcVnVector3_SINT.TcPOU, Node_ContainerType_Vector_TcVnVector2_REAL.TcPOU, Node_ContainerType_Vector_TcVnVector2_DINT.TcPOU, Node_ContainerType_Vector_TcVnVector2_UINT.TcPOU, Node_ContainerType_Vector_TcVnVector2_INT.TcPOU, Node_ContainerType_Vector_TcVnVector2_USINT.TcPOU, Node_ContainerType_Vector_TcVnVector2_SINT.TcPOU, Node_ContainerType_Vector_Vector_LREAL.TcPOU, Node_ContainerType_Vector_Vector_REAL.TcPOU, Node_ContainerType_Vector_Vector_ULINT.TcPOU, Node_ContainerType_Vector_Vector_UDINT.TcPOU, Node_ContainerType_Vector_Vector_TcVnPoint3_REAL.TcPOU, Node_ContainerType_Vector_Vector_TcVnPoint2_REAL.TcPOU, Node_ContainerType_Vector_Vector_TcVnPoint2_DINT.TcPOU, Node_ContainerType_Vector_TcVnPoint3_LREAL.TcPOU, Node_ContainerType_Vector_TcVnPoint3_REAL.TcPOU, Node_ContainerType_Vector_TcVnPoint2_LREAL.TcPOU, Node_ContainerType_Vector_TcVnPoint2_REAL.TcPOU, Node_ContainerType_Vector_TcVnPoint2_DINT.TcPOU, Node_ContainerType_Vector_ITcVnImage.TcPOU, Node_ContainerType_Vector_LREAL.TcPOU, Node_ContainerType_Vector_REAL.TcPOU, Node_ContainerType_Vector_ULINT.TcPOU, Node_ContainerType_Vector_SINT.TcPOU, Node_ContainerType_Vector_DINT.TcPOU, Node_ContainerType_Vector_UDINT.TcPOU, Node_ContainerType_Vector_USINT.TcPOU, Node_ContainerType_Vector_INT.TcPOU, Node_RGBA_RANDOM.TcPOU, Node_RGBA_BLUE.TcPOU, Node_RGBA_MAGENTA.TcPOU, Node_RGBA_CYAN.TcPOU, Node_RGBA_YELLOW.TcPOU, Node_RGBA_WHITE.TcPOU, Node_RGBA_RED.TcPOU, Node_RGBA_GREEN.TcPOU, Node_RGBA_BLACK.TcPOU
//   Nodes/Container Statistics/MaxElementwise/ Node_F_VN_MaxElementElementwise_DINT.TcPOU (not stored), Node_F_VN_MaxElementElementwise_INT.TcPOU (not stored), Node_F_VN_MaxElementElementwise_LREAL.TcPOU (not stored), Node_F_VN_MaxElementElementwise_REAL.TcPOU (not stored), Node_F_VN_MaxElementElementwise_SINT.TcPOU (not stored), Node_F_VN_MaxElementElementwise_TcVnPoint2_DINT.TcPOU (not stored), Node_F_VN_MaxElementElementwise_TcVnPoint2_LREAL.TcPOU (not stored), Node_F_VN_MaxElementElementwise_TcVnPoint2_REAL.TcPOU (not stored), Node_F_VN_MaxElementElementwise_TcVnPoint3_LREAL.TcPOU (not stored), Node_F_VN_MaxElementElementwise_TcVnPoint3_REAL.TcPOU (not stored), Node_F_VN_MaxElementElementwise_TcVnVector2_DINT.TcPOU (not stored), Node_F_VN_MaxElementElementwise_TcVnVector2_INT.TcPOU (not stored), Node_F_VN_MaxElementElementwise_TcVnVector2_REAL.TcPOU (not stored), Node_F_VN_MaxElementElementwise_TcVnVector2_SINT.TcPOU (not stored), Node_F_VN_MaxElementElementwise_TcVnVector2_UINT.TcPOU (not stored), Node_F_VN_MaxElementElementwise_TcVnVector2_USINT.TcPOU (not stored), Node_F_VN_MaxElementElementwise_TcVnVector3_INT.TcPOU (not stored), Node_F_VN_MaxElementElementwise_TcVnVector3_REAL.TcPOU (not stored), Node_F_VN_MaxElementElementwise_TcVnVector3_SINT.TcPOU (not stored), Node_F_VN_MaxElementElementwise_TcVnVector3_UINT.TcPOU (not stored), Node_F_VN_MaxElementElementwise_TcVnVector3_USINT.TcPOU (not stored), Node_F_VN_MaxElementElementwise_TcVnVector4_DINT.TcPOU (not stored), Node_F_VN_MaxElementElementwise_TcVnVector4_INT.TcPOU (not stored), Node_F_VN_MaxElementElementwise_TcVnVector4_LREAL.TcPOU (not stored), Node_F_VN_MaxElementElementwise_TcVnVector4_REAL.TcPOU (not stored), Node_F_VN_MaxElementElementwise_TcVnVector4_SINT.TcPOU (not stored), Node_F_VN_MaxElementElementwise_TcVnVector4_UINT.TcPOU (not stored), Node_F_VN_MaxElementElementwise_TcVnVector4_USINT.TcPOU (not stored), Node_F_VN_MaxElementElementwise_UDINT.TcPOU (not stored), Node_F_VN_MaxElementElementwise_UINT.TcPOU (not stored), Node_F_VN_MaxElementElementwise_ULINT.TcPOU (not stored), Node_F_VN_MaxElementElementwise_USINT.TcPOU (not stored)
//   Nodes/Container Statistics/MedianElementwise/ Node_F_VN_MedianElementElementwise_DINT.TcPOU (not stored), Node_F_VN_MedianElementElementwise_INT.TcPOU (not stored), Node_F_VN_MedianElementElementwise_LREAL.TcPOU (not stored), Node_F_VN_MedianElementElementwise_REAL.TcPOU (not stored), Node_F_VN_MedianElementElementwise_SINT.TcPOU (not stored), Node_F_VN_MedianElementElementwise_TcVnPoint2_DINT.TcPOU (not stored), Node_F_VN_MedianElementElementwise_TcVnPoint2_LREAL.TcPOU (not stored), Node_F_VN_MedianElementElementwise_TcVnPoint2_REAL.TcPOU (not stored), Node_F_VN_MedianElementElementwise_TcVnPoint3_LREAL.TcPOU (not stored), Node_F_VN_MedianElementElementwise_TcVnPoint3_REAL.TcPOU (not stored), Node_F_VN_MedianElementElementwise_TcVnVector2_DINT.TcPOU (not stored), Node_F_VN_MedianElementElementwise_TcVnVector2_INT.TcPOU (not stored), Node_F_VN_MedianElementElementwise_TcVnVector2_REAL.TcPOU (not stored), Node_F_VN_MedianElementElementwise_TcVnVector2_SINT.TcPOU (not stored), Node_F_VN_MedianElementElementwise_TcVnVector2_UINT.TcPOU (not stored), Node_F_VN_MedianElementElementwise_TcVnVector2_USINT.TcPOU (not stored), Node_F_VN_MedianElementElementwise_TcVnVector3_INT.TcPOU (not stored), Node_F_VN_MedianElementElementwise_TcVnVector3_REAL.TcPOU (not stored), Node_F_VN_MedianElementElementwise_TcVnVector3_SINT.TcPOU (not stored), Node_F_VN_MedianElementElementwise_TcVnVector3_UINT.TcPOU (not stored), Node_F_VN_MedianElementElementwise_TcVnVector3_USINT.TcPOU (not stored), Node_F_VN_MedianElementElementwise_TcVnVector4_DINT.TcPOU (not stored), Node_F_VN_MedianElementElementwise_TcVnVector4_INT.TcPOU (not stored), Node_F_VN_MedianElementElementwise_TcVnVector4_LREAL.TcPOU (not stored), Node_F_VN_MedianElementElementwise_TcVnVector4_REAL.TcPOU (not stored), Node_F_VN_MedianElementElementwise_TcVnVector4_SINT.TcPOU (not stored), Node_F_VN_MedianElementElementwise_TcVnVector4_UINT.TcPOU (not stored), Node_F_VN_MedianElementElementwise_TcVnVector4_USINT.TcPOU (not stored), Node_F_VN_MedianElementElementwise_UDINT.TcPOU (not stored), Node_F_VN_MedianElementElementwise_UINT.TcPOU (not stored), Node_F_VN_MedianElementElementwise_ULINT.TcPOU (not stored), Node_F_VN_MedianElementElementwise_USINT.TcPOU (not stored)
//   Nodes/Container Statistics/MinElementwise/ Node_F_VN_MinElementElementwise_DINT.TcPOU (not stored), Node_F_VN_MinElementElementwise_INT.TcPOU (not stored), Node_F_VN_MinElementElementwise_LREAL.TcPOU (not stored), Node_F_VN_MinElementElementwise_REAL.TcPOU (not stored), Node_F_VN_MinElementElementwise_SINT.TcPOU (not stored), Node_F_VN_MinElementElementwise_TcVnPoint2_DINT.TcPOU (not stored), Node_F_VN_MinElementElementwise_TcVnPoint2_LREAL.TcPOU (not stored), Node_F_VN_MinElementElementwise_TcVnPoint2_REAL.TcPOU (not stored), Node_F_VN_MinElementElementwise_TcVnPoint3_LREAL.TcPOU (not stored), Node_F_VN_MinElementElementwise_TcVnPoint3_REAL.TcPOU (not stored), Node_F_VN_MinElementElementwise_TcVnVector2_DINT.TcPOU (not stored), Node_F_VN_MinElementElementwise_TcVnVector2_INT.TcPOU (not stored), Node_F_VN_MinElementElementwise_TcVnVector2_REAL.TcPOU (not stored), Node_F_VN_MinElementElementwise_TcVnVector2_SINT.TcPOU (not stored), Node_F_VN_MinElementElementwise_TcVnVector2_UINT.TcPOU (not stored), Node_F_VN_MinElementElementwise_TcVnVector2_USINT.TcPOU (not stored), Node_F_VN_MinElementElementwise_TcVnVector3_INT.TcPOU (not stored), Node_F_VN_MinElementElementwise_TcVnVector3_REAL.TcPOU (not stored), Node_F_VN_MinElementElementwise_TcVnVector3_SINT.TcPOU (not stored), Node_F_VN_MinElementElementwise_TcVnVector3_UINT.TcPOU (not stored), Node_F_VN_MinElementElementwise_TcVnVector3_USINT.TcPOU (not stored), Node_F_VN_MinElementElementwise_TcVnVector4_DINT.TcPOU (not stored), Node_F_VN_MinElementElementwise_TcVnVector4_INT.TcPOU (not stored), Node_F_VN_MinElementElementwise_TcVnVector4_LREAL.TcPOU (not stored), Node_F_VN_MinElementElementwise_TcVnVector4_REAL.TcPOU (not stored), Node_F_VN_MinElementElementwise_TcVnVector4_SINT.TcPOU (not stored), Node_F_VN_MinElementElementwise_TcVnVector4_UINT.TcPOU (not stored), Node_F_VN_MinElementElementwise_TcVnVector4_USINT.TcPOU (not stored), Node_F_VN_MinElementElementwise_UDINT.TcPOU (not stored), Node_F_VN_MinElementElementwise_UINT.TcPOU (not stored), Node_F_VN_MinElementElementwise_ULINT.TcPOU (not stored), Node_F_VN_MinElementElementwise_USINT.TcPOU (not stored)
//   Nodes/Container Statistics/ Node_F_VN_ContainerAverage.TcPOU, Node_F_VN_ContainerAverageElementwise3.TcPOU, Node_F_VN_ContainerAverageElementwise4.TcPOU, Node_F_VN_ContainerAverageVarianceElementwise2.TcPOU, Node_F_VN_ContainerAverageVariance.TcPOU, Node_F_VN_ContainerAverageElementwise2.TcPOU, Node_F_VN_ContainerAverageVarianceElementwise3.TcPOU, Node_F_VN_ContainerAverageVarianceElementwise4.TcPOU, Node_F_VN_MaxElement.TcPOU, Node_F_VN_MinElement.TcPOU, Node_F_VN_MedianElement.TcPOU
//   Nodes/Contour Analysis/ Node_F_VN_ApproximatePolygon.TcPOU, Node_F_VN_ContourCircularityExp.TcPOU, Node_F_VN_FitLineExp.TcPOU, Node_F_VN_MatchContours1vsN.TcPOU, Node_F_VN_ContourElongation.TcPOU, Node_F_VN_ContourOrientationExp.TcPOU, Node_F_VN_ContourExtremePoint.TcPOU, Node_F_VN_MatchContours1vsNExp.TcPOU, Node_F_VN_UprightBoundingRectangle.TcPOU, Node_F_VN_ContourPerimeter.TcPOU, Node_F_VN_ContourInertiaRatio.TcPOU, Node_F_VN_ContourCircularity.TcPOU, Node_F_VN_ContourCenterOfMass.TcPOU, Node_F_VN_ContourConvexity.TcPOU, Node_F_VN_ContourEccentricity.TcPOU, Node_F_VN_CheckIfPointIsInsideContour.TcPOU, Node_F_VN_ContourRoundness.TcPOU, Node_F_VN_ContourOrientation.TcPOU, Node_F_VN_ContourArea.TcPOU, Node_F_VN_ConvexHullPoints.TcPOU, Node_F_VN_ConvexHullPointsExp.TcPOU, Node_F_VN_ConvexityDefects.TcPOU, Node_F_VN_EnclosingRectangle.TcPOU, Node_F_VN_EnclosingTriangle.TcPOU, Node_F_VN_FitLine.TcPOU, Node_F_VN_EnclosingCircle.TcPOU, Node_F_VN_ContourMoments.TcPOU, Node_F_VN_FitEllipse.TcPOU, Node_F_VN_MatchContours.TcPOU, Node_F_VN_MatchContoursExp.TcPOU
//   Nodes/Drawing/ Node_F_VN_DrawArrowExp.TcPOU, Node_F_VN_DrawArrowExp_TcVnVector4_DINT.TcPOU, Node_F_VN_DrawArrow_TcVnVector4_DINT.TcPOU, Node_F_VN_DrawCircleExp.TcPOU, Node_F_VN_DrawCircles.TcPOU, Node_F_VN_DrawCirclesExp.TcPOU, Node_F_VN_DrawCircularArcExp.TcPOU, Node_F_VN_DrawComponentsExp.TcPOU, Node_F_VN_DrawContoursExp.TcPOU, Node_F_VN_DrawEllipseExp.TcPOU, Node_F_VN_DrawArrow.TcPOU, Node_F_VN_DrawComponents.TcPOU, Node_F_VN_DrawKeypointsExp.TcPOU, Node_F_VN_DrawMatches.TcPOU, Node_F_VN_DrawLineExp.TcPOU, Node_F_VN_DrawLineExp_TcVnVector4_DINT.TcPOU, Node_F_VN_DrawLineExp_TcVnVector4_LREAL.TcPOU, Node_F_VN_DrawLines.TcPOU, Node_F_VN_DrawLinesExp.TcPOU, Node_F_VN_DrawMatchesExp.TcPOU, Node_F_VN_DrawOrientation.TcPOU, Node_F_VN_DrawCircularArc.TcPOU, Node_F_VN_DrawOrientationExp.TcPOU, Node_F_VN_DrawPoints.TcPOU, Node_F_VN_DrawPointExp.TcPOU, Node_F_VN_DrawPointsExp.TcPOU, Node_F_VN_DrawPolygonExp.TcPOU, Node_F_VN_FillEllipse.TcPOU, Node_F_VN_DrawKeypoints.TcPOU, Node_F_VN_DrawLine_TcVnVector4_DINT.TcPOU, Node_F_VN_DrawPolygon.TcPOU, Node_F_VN_DrawRectangle_TcVnRectangle_DINT.TcPOU, Node_F_VN_DrawRectangle_TcVnRectangle_UDINT.TcPOU, Node_F_VN_DrawRotatedRectangleExp.TcPOU, Node_F_VN_DrawEllipse.TcPOU, Node_F_VN_FillPolygon.TcPOU, Node_F_VN_FillContours.TcPOU, Node_F_VN_DrawRotatedRectangle.TcPOU, Node_F_VN_FillRotatedRectangle.TcPOU, Node_F_VN_PlotIntensityProfile.TcPOU, Node_F_VN_DrawRectangle.TcPOU, Node_F_VN_FillRectangle.TcPOU, Node_F_VN_FillCircle.TcPOU, Node_F_VN_DrawContours.TcPOU, Node_F_VN_DrawLine.TcPOU, Node_F_VN_DrawCircle.TcPOU, Node_F_VN_DrawPoint.TcPOU, Node_F_VN_DrawLine_TcVnVector4_LREAL.TcPOU, Node_F_VN_PlotIntensityProfileExp.TcPOU, Node_F_VN_PutLabel.TcPOU, Node_F_VN_PutLabelExp.TcPOU, Node_F_VN_PutText.TcPOU, Node_F_VN_PutTextExp.TcPOU
//   Nodes/Fourier Analysis/ Node_F_VN_CreateBandrejectButterworthFilter.TcPOU, Node_F_VN_CreateBandpassGaussianFilter.TcPOU, Node_F_VN_CreateBandrejectGaussianFilter.TcPOU, Node_F_VN_CreateHighpassButterworthFilter.TcPOU, Node_F_VN_CreateBandpassButterworthFilter.TcPOU, Node_F_VN_CreateLowpassGaussianFilter.TcPOU, Node_F_VN_CreateHighpassGaussianFilter.TcPOU, Node_F_VN_CreateLowpassButterworthFilter.TcPOU, Node_F_VN_OptimalDftSize.TcPOU, Node_F_VN_InverseDft.TcPOU, Node_F_VN_Dft.TcPOU
//   Nodes/Geometric and Coord Transform/Calibration/ Node_F_VN_CalibrateCameraPlanar.TcPOU (not stored), Node_F_VN_GenerateCalibrationPatternReferencePoints.TcPOU (not stored), Node_F_VN_SolvePnP.TcPOU (not stored), Node_F_VN_CompensateLensDistortion.TcPOU (not stored), Node_F_VN_CompensateLensDistortionExp1.TcPOU (not stored), Node_F_VN_CompensateLensDistortionExp2.TcPOU (not stored), Node_F_VN_CompensateLensDistortionForPointsExp2.TcPOU (not stored), Node_F_VN_CompensateLensDistortionForPoints.TcPOU (not stored), Node_F_VN_CompensateLensDistortionForPointsExp1.TcPOU (not stored), Node_F_VN_CalibrateCamera.TcPOU (not stored), Node_F_VN_SolvePnPExp.TcPOU (not stored), Node_F_VN_SortDetectedPatternPoints.TcPOU (not stored), Node_F_VN_DetectPatternPoints.TcPOU (not stored), Node_F_VN_CalibrateCameraManually.TcPOU (not stored), Node_F_VN_CalibrateCameraManuallyExp.TcPOU (not stored), Node_F_VN_CalibrateCameraPlanarExp.TcPOU (not stored), Node_F_VN_DetectPatternPointsExp.TcPOU (not stored), Node_F_VN_ImagePointsWorldDistance.TcPOU (not stored), Node_F_VN_TransformCoordinatesImageToWorld_Container.TcPOU (not stored), Node_F_VN_TransformCoordinatesImageToWorld_Point.TcPOU (not stored), Node_F_VN_TransformCoordinatesPlanar_Container.TcPOU (not stored), Node_F_VN_TransformCoordinatesPlanar_Point.TcPOU (not stored), Node_F_VN_TransformCoordinatesWorldToImage_Container.TcPOU (not stored), Node_F_VN_TransformCoordinatesWorldToImage_Point.TcPOU (not stored), Node_F_VN_DetectPatternPoints2.TcPOU (not stored), Node_F_VN_SortAxisAlignedPatternPoints.TcPOU (not stored)
//   Nodes/Geometric and Coord Transform/ Node_F_VN_DecomposeHomography.TcPOU, Node_F_VN_DecomposeHomographyExp.TcPOU, Node_F_VN_ResizeRegion_TcVnRectangle_DINT.TcPOU, Node_F_VN_ApplyRotationToAffineTransformationExp.TcPOU, Node_F_VN_ApplyScalingToAffineTransformation.TcPOU, Node_F_VN_ApplyScalingToAffineTransformationExp.TcPOU, Node_F_VN_ApplyTranslationToAffineTransformationExp.TcPOU, Node_F_VN_ApplyTranslationToAffineTransformation.TcPOU, Node_F_VN_ApplyYAxisInversionToAffineTransformation.TcPOU, Node_F_VN_AlignRotatedImageRegion.TcPOU, Node_F_VN_ApplyRotationToAffineTransformation.TcPOU, Node_F_VN_ConvertCartesianToPolarAnglesExp.TcPOU, Node_F_VN_ConvertCartesianToPolarMagnitudes.TcPOU, Node_F_VN_ConvertCartesianToPolarPoints.TcPOU, Node_F_VN_ConvertCartesianToPolarPointsExp.TcPOU, Node_F_VN_ConvertPolarToCartesianPoints.TcPOU, Node_F_VN_ConvertPolarToCartesianPointsExp.TcPOU, Node_F_VN_DecomposeAffineTransformationExp.TcPOU, Node_F_VN_GenerateAffineTransformationUnitMatrix2D.TcPOU, Node_F_VN_DecomposeAffineTransformation.TcPOU, Node_F_VN_GetAffineTransformation2D.TcPOU, Node_F_VN_GetPerspectiveTransformation.TcPOU, Node_F_VN_Homography.TcPOU, Node_F_VN_HomographyExp.TcPOU, Node_F_VN_RemapImageToLogPolarSpace.TcPOU, Node_F_VN_RemapImageToPolarSpace.TcPOU, Node_F_VN_ResizeImageExp.TcPOU, Node_F_VN_RotateImage.TcPOU, Node_F_VN_ResizeImage.TcPOU, Node_F_VN_RotateImageExp.TcPOU, Node_F_VN_RotateImageExp2.TcPOU, Node_F_VN_WarpAffine.TcPOU, Node_F_VN_PyramidDown.TcPOU, Node_F_VN_FlipImage.TcPOU, Node_F_VN_ApplyYAxisInversionToAffineTransformationExp.TcPOU, Node_F_VN_PyramidUp.TcPOU, Node_F_VN_InvertAffineTransformation.TcPOU, Node_F_VN_GetAffineTransformation.TcPOU, Node_F_VN_WarpAffineExp.TcPOU, Node_F_VN_WarpPerspectiveExp.TcPOU, Node_F_VN_WarpAffine_Container.TcPOU, Node_F_VN_PerspectiveTransformation.TcPOU, Node_F_VN_ConvertCartesianToPolarAngles.TcPOU, Node_F_VN_WarpPerspective_Rectangle.TcPOU, Node_F_VN_WarpPerspective_Point.TcPOU, Node_F_VN_WarpPerspective_Container.TcPOU, Node_F_VN_WarpAffine_Rectangle.TcPOU, Node_F_VN_WarpAffine_Point.TcPOU, Node_F_VN_WarpPerspective.TcPOU, Node_F_VN_ConvertCartesianToPolarAngleImage.TcPOU, Node_F_VN_ConvertCartesianToPolarAngleImageExp.TcPOU, Node_F_VN_ConvertCartesianToPolarImages.TcPOU, Node_F_VN_ConvertCartesianToPolarImagesExp.TcPOU, Node_F_VN_ConvertCartesianToPolarMagnitudeImage.TcPOU, Node_F_VN_ConvertPolarToCartesianImages.TcPOU, Node_F_VN_ConvertPolarToCartesianImagesExp.TcPOU, Node_F_VN_ConvertMaps.TcPOU, Node_F_VN_RemapImage.TcPOU, Node_F_VN_RemapImageExp.TcPOU, Node_F_VN_RemapImageToLogPolarSpaceExp.TcPOU, Node_F_VN_RemapImageToLogPolarSpaceExp2.TcPOU, Node_F_VN_RemapImageToPolarSpaceExp.TcPOU, Node_F_VN_RemapImageToPolarSpaceExp2.TcPOU, Node_F_VN_AlignRotatedImageRegionExp.TcPOU
//   Nodes/Helpers/ Node_Mux10Way_ITcVnImage.TcPOU
//   Nodes/Image Analysis/ Node_F_VN_CannyEdgeDetectionExp.TcPOU, Node_F_VN_ConnectedComponentsExp.TcPOU, Node_F_VN_ConnectedComponentsWithStatsExp.TcPOU, Node_F_VN_ConnectedComponentsWithStats.TcPOU, Node_F_VN_GetConnectedComponent.TcPOU, Node_F_VN_GetConnectedComponentExp.TcPOU, Node_F_VN_UprightInnerRectangle.TcPOU, Node_F_VN_CountNonZeroPixels.TcPOU, Node_F_VN_DistanceTransformation.TcPOU, Node_F_VN_ConnectedComponents.TcPOU, Node_F_VN_DistanceTransformationExp.TcPOU, Node_F_VN_ImageAverage.TcPOU, Node_F_VN_ImageAverageStdDev.TcPOU, Node_F_VN_ImageAverageExp.TcPOU, Node_F_VN_ImageAverageStdDevExp.TcPOU, Node_F_VN_CannyEdgeDetection.TcPOU, Node_F_VN_ImageCenterOfMass.TcPOU, Node_F_VN_ImageCenterOfMassExp.TcPOU, Node_F_VN_RegionOrientation.TcPOU, Node_F_VN_ImageMedianExp.TcPOU, Node_F_VN_ImageMoments.TcPOU, Node_F_VN_ImageMedian.TcPOU, Node_F_VN_MaxPixelValue.TcPOU, Node_F_VN_MaxPixelValueExp.TcPOU, Node_F_VN_MinPixelValueExp.TcPOU, Node_F_VN_MinPixelValue.TcPOU, Node_F_VN_RegionOrientationExp.TcPOU, Node_F_VN_ImageAbsoluteAverage.TcPOU, Node_F_VN_UprightInnerRectangleExp.TcPOU
//   Nodes/Image Analysis/Object Detection/ Node_F_VN_DetectBlobs.TcPOU (not stored), Node_F_VN_DetectBlobsExp.TcPOU (not stored), Node_F_VN_FindContours.TcPOU (not stored), Node_F_VN_FindContoursExp.TcPOU (not stored), Node_F_VN_FindTemplateWalshExp.TcPOU (not stored), Node_F_VN_FindTemplateWalshExp_AngleRange.TcPOU (not stored), Node_F_VN_FindTemplateWalsh_AngleRange.TcPOU (not stored), Node_F_VN_HoughCircles.TcPOU (not stored), Node_F_VN_HoughCirclesExp.TcPOU (not stored), Node_F_VN_MatchImageHuMoments.TcPOU (not stored), Node_F_VN_HoughLines.TcPOU (not stored), Node_F_VN_HoughLinesP.TcPOU (not stored), Node_F_VN_HoughLinesPExp.TcPOU (not stored), Node_F_VN_FindContourHierarchyExp.TcPOU (not stored), Node_F_VN_MatchTemplate.TcPOU (not stored), Node_F_VN_MatchTemplateAndEvaluate.TcPOU (not stored), Node_F_VN_MatchTemplateWalshExp.TcPOU (not stored), Node_F_VN_MatchTemplateWalsh.TcPOU (not stored), Node_F_VN_FindTemplateWalsh.TcPOU (not stored), Node_F_VN_SalientFeatures.TcPOU (not stored), Node_F_VN_FindRois.TcPOU (not stored), Node_F_VN_MergeRegions.TcPOU (not stored), Node_F_VN_MatchTemplateExp.TcPOU (not stored), Node_F_VN_MatchTemplateAndEvaluateExp.TcPOU (not stored)
//   Nodes/Image Color and Contrast Processing/ Node_F_VN_ApplyColorMap.TcPOU, Node_F_VN_Clahe.TcPOU, Node_F_VN_ClaheExp.TcPOU, Node_F_VN_GenerateCustomColorMap.TcPOU, Node_F_VN_HistogramExp.TcPOU, Node_F_VN_ReferenceColorSimilarity_TcVnVector3_LREAL.TcPOU, Node_F_VN_Histogram.TcPOU, Node_F_VN_HistogramEqualization.TcPOU, Node_F_VN_HistogramEqualizationExp.TcPOU, Node_F_VN_InvertImageColor.TcPOU, Node_F_VN_ConvertColorSpace.TcPOU, Node_F_VN_GenerateColorMap.TcPOU, Node_F_VN_NormalizeImage.TcPOU, Node_F_VN_NormalizeImageForDisplay.TcPOU, Node_F_VN_ReferenceColorSimilarityExp_TcVnVector3_LREAL.TcPOU, Node_F_VN_WhiteBalance.TcPOU, Node_F_VN_InvertImageColorExp.TcPOU, Node_F_VN_NormalizeImageExp.TcPOU
//   Nodes/Image Filtering/ Node_F_VN_BilateralFilter.TcPOU, Node_F_VN_BoxFilterExp.TcPOU, Node_F_VN_GaussianFilterExp.TcPOU, Node_F_VN_LaplacianFilterExp.TcPOU, Node_F_VN_ScharrFilter.TcPOU, Node_F_VN_CreateStructuringElement.TcPOU, Node_F_VN_RemoveLocalMaxima.TcPOU, Node_F_VN_MedianFilter.TcPOU, Node_F_VN_MorphologicalOperator.TcPOU, Node_F_VN_RemoveLocalMinima.TcPOU, Node_F_VN_ScharrFilterExp.TcPOU, Node_F_VN_BilateralFilterExp.TcPOU, Node_F_VN_SobelFilterExp.TcPOU, Node_F_VN_SobelFilter.TcPOU, Node_F_VN_VarianceFilter.TcPOU, Node_F_VN_LocalMaxima.TcPOU, Node_F_VN_DarkBorderObjects.TcPOU, Node_F_VN_FillHoles.TcPOU, Node_F_VN_BoxFilter.TcPOU, Node_F_VN_BrightBorderObjects.TcPOU, Node_F_VN_GaussianFilter.TcPOU, Node_F_VN_LaplacianFilter.TcPOU, Node_F_VN_LocalMinima.TcPOU, Node_F_VN_VarianceFilterExp.TcPOU
//   Nodes/Image Segmentation/ Node_F_VN_AdaptiveThresholdExp.TcPOU, Node_F_VN_SauvolaThreshold.TcPOU, Node_F_VN_DoubleThreshold.TcPOU, Node_F_VN_WatershedSegmentationExp.TcPOU, Node_F_VN_CheckColorRange.TcPOU, Node_F_VN_AdaptiveThreshold.TcPOU, Node_F_VN_Threshold.TcPOU
//   Nodes/Keypoint Features/ Node_F_VN_FilterGoodMatches.TcPOU, Node_F_VN_FindReferenceKeyPointsInImage.TcPOU, Node_F_VN_FindReferenceKeyPointsInImageExp.TcPOU, Node_F_VN_FindReferenceKeyPointsInImageAKAZE.TcPOU, Node_F_VN_FindReferenceKeyPointsInImageAKAZEExp.TcPOU, Node_F_VN_FindReferenceKeyPointsInImageBRISK.TcPOU, Node_F_VN_FindReferenceKeyPointsInImageBRISKExp.TcPOU, Node_F_VN_FindReferenceKeyPointsInImageORB.TcPOU, Node_F_VN_FindReferenceKeyPointsInImageORBExp.TcPOU, Node_F_VN_KeyPointsAGAST.TcPOU, Node_F_VN_KeyPointsAGASTExp.TcPOU, Node_F_VN_GetMatchCoordinates.TcPOU, Node_F_VN_KeyPointsAndDescriptorsAKAZE.TcPOU, Node_F_VN_KeyPointsAndDescriptorsAKAZEExp.TcPOU, Node_F_VN_KeyPointsAndDescriptorsBRISKExp.TcPOU, Node_F_VN_KeyPointsAndDescriptorsBRISK.TcPOU, Node_F_VN_KeyPointsAndDescriptorsKAZEExp.TcPOU, Node_F_VN_KeyPointsAndDescriptorsKAZE.TcPOU, Node_F_VN_KeyPointsAndDescriptorsORBExp.TcPOU, Node_F_VN_KeyPointsAndDescriptorsORB.TcPOU, Node_F_VN_KeyPointsFASTExp.TcPOU, Node_F_VN_MatchDescriptorsBF.TcPOU (not stored), Node_F_VN_KeyPointsGFTTExp.TcPOU, Node_F_VN_KeyPointsGFTT.TcPOU, Node_F_VN_KeyPointsFAST.TcPOU, Node_F_VN_KeyPointsMSERExp.TcPOU, Node_F_VN_KeyPointsMSER.TcPOU, Node_F_VN_KeyPointsSBExp.TcPOU, Node_F_VN_MatchDescriptorsFlannLsh.TcPOU (not stored), Node_F_VN_MatchDescriptorsFlannLshExp.TcPOU (not stored), Node_F_VN_MatchDescriptorsKnnBF.TcPOU (not stored), Node_F_VN_MatchDescriptorsKnnFlannLsh.TcPOU (not stored), Node_F_VN_MatchDescriptorsKnnFlannLshExp.TcPOU (not stored), Node_F_VN_RegionsMSER.TcPOU (not stored), Node_F_VN_KeyPointsSB.TcPOU, Node_F_VN_RegionsMSERExp.TcPOU (not stored), Node_F_VN_MatchDescriptorsBFExp.TcPOU (not stored), Node_F_VN_MatchDescriptorsKnnBFExp.TcPOU (not stored)
//   Nodes/Measurement/ Node_F_VN_LocateEdge.TcPOU (not stored), Node_F_VN_LocateEdges.TcPOU (not stored), Node_F_VN_LocateEdgeExp.TcPOU (not stored), Node_F_VN_LocateEdgesExp.TcPOU (not stored), Node_F_VN_AdjustSearchWindowOrientationToLinearEdge.TcPOU (not stored), Node_F_VN_LocateCircularArc.TcPOU (not stored), Node_F_VN_ClosestPointsBF.TcPOU (not stored), Node_F_VN_LocateEllipseExp.TcPOU (not stored), Node_F_VN_MeasureAngleBetweenEdges.TcPOU (not stored), Node_F_VN_LocateEllipse.TcPOU (not stored), Node_F_VN_MeasureEdgeDistance.TcPOU (not stored), Node_F_VN_MeasureEdgeDistanceExp.TcPOU (not stored), Node_F_VN_MeasureMinEdgeDistance.TcPOU (not stored), Node_F_VN_LocateAxisAlignedEdges.TcPOU (not stored), Node_F_VN_LocateAxisAlignedEdgesExp.TcPOU (not stored), Node_F_VN_LocateCircularArcExp.TcPOU (not stored), Node_F_VN_LocateCircularArcExp2.TcPOU (not stored), Node_F_VN_LocateEdgeExp2.TcPOU (not stored), Node_F_VN_LocateEdgesExp2.TcPOU (not stored), Node_F_VN_LocateEllipseExp2.TcPOU (not stored), Node_F_VN_MeasureAngleBetweenEdgesExp.TcPOU (not stored), Node_F_VN_MeasureAngleBetweenEdgesExp2.TcPOU (not stored), Node_F_VN_MeasureEdgeDistanceExp2.TcPOU (not stored), Node_F_VN_MeasureMinEdgeDistanceExp.TcPOU (not stored), Node_F_VN_MeasureMinEdgeDistanceExp2.TcPOU (not stored)
//   Nodes/Miscellaneous/ Node_FB_VN_InitializeFunction.TcPOU (not stored) (excluded from build), Node_F_VN_DeinitializeFunction.TcPOU (not stored), Node_F_VN_ClipLineToBoundary_ITcVnImage.TcPOU (not stored), Node_F_VN_ClipLineToBoundary_TcVnRectangle_DINT.TcPOU (not stored), Node_F_VN_CheckFunctionInitialization.TcPOU (not stored), Node_F_VN_OrthogonalVector_TcVnVector2_LREAL.TcPOU (not stored), Node_F_VN_OrthogonalVector_TcVnVector2_REAL.TcPOU (not stored), Node_F_VN_PointToLineDistance_TcVnPoint2_DINT.TcPOU (not stored), Node_F_VN_OrthogonalVector_TcVnVector2_DINT.TcPOU (not stored), Node_F_VN_PointToPointDirection_TcVnPoint2_LREAL.TcPOU (not stored), Node_F_VN_PointToPointDirection_TcVnPoint2_REAL.TcPOU (not stored), Node_F_VN_PointToPointDistance_TcVnPoint2_DINT.TcPOU (not stored), Node_F_VN_PointToLineDistance_TcVnPoint2_LREAL.TcPOU (not stored), Node_F_VN_PointToLineDistance_TcVnPoint2_REAL.TcPOU (not stored), Node_F_VN_PointToPointDirection_TcVnPoint2_DINT.TcPOU (not stored), Node_F_VN_PointToPointDistance_TcVnPoint2_LREAL.TcPOU (not stored), Node_F_VN_PointToPointDistance_TcVnPoint2_REAL.TcPOU (not stored), Node_F_VN_RotatedRectangleCorners.TcPOU (not stored), Node_F_VN_HuMomentInvariants.TcPOU (not stored), Node_F_VN_InvertMatrix3x3.TcPOU (not stored), Node_F_VN_ClipLineToBoundary.TcPOU (not stored), Node_F_VN_MultiplyMatrices.TcPOU (not stored) (excluded from build), Node_F_VN_LineIntersectionPoint.TcPOU (not stored), Node_F_VN_LineIntersectionPointAndAngle.TcPOU (not stored), Node_F_VN_RotatedRectangleIntersection.TcPOU (not stored)
//   Nodes/Neural Network/ Node_F_VN_ReduceArg.TcPOU (not stored), Node_F_VN_Sigmoid.TcPOU (not stored), Node_F_VN_SigmoidExp.TcPOU (not stored), Node_F_VN_Reduce.TcPOU (not stored), Node_F_VN_SoftMax.TcPOU (not stored)
//   Nodes/OCR/ Node_F_VN_OCR.TcPOU (not stored), Node_F_VN_OCRExp.TcPOU (not stored)
//   Nodes/Texture Analysis/ Node_F_VN_HaralickFeatures.TcPOU (not stored), Node_F_VN_Granulometry.TcPOU (not stored)
//   Nodes/ VisionNodePack.TcPOU
//   Nodes/VisionNode/ VisionNode.TcPOU (not stored), VisionHardwareNode.TcPOU (not stored)
//   Nodes/Polarization/ Node_F_VN_DemosaicPolarizedImage.TcPOU (not stored), Node_F_VN_AngleAndDegreeOfLinearPolarization.TcPOU (not stored), Node_F_VN_PolarizedImageGlareReduction.TcPOU (not stored)

// ---- GVL_COLOURS.TcGVL
{attribute 'qualified_only'}
VAR_GLOBAL
    RGBA_BLACK    : TcVnVector4_LREAL := [0, 0, 0, 255];
    RGBA_RED      : TcVnVector4_LREAL := [255, 0, 0, 255];
    RGBA_YELLOW   : TcVnVector4_LREAL := [255, 255, 0, 255];
    RGBA_GREEN    : TcVnVector4_LREAL := [0, 255, 0, 255];
    RGBA_CYAN     : TcVnVector4_LREAL := [0, 255, 255, 255];
    RGBA_BLUE     : TcVnVector4_LREAL := [0, 0, 255, 255];
    RGBA_MAGENTA  : TcVnVector4_LREAL := [255, 0, 255, 255];
    RGBA_WHITE    : TcVnVector4_LREAL := [255, 255, 255, 255];
    RGBA_RANDOM   : TcVnVector4_LREAL := [-1, -1, -1, -1];
END_VAR

// ---- Datatypes/Aliases/_GVCP_REGISTER_ADDRESS.TcPOU
{attribute 'linkalways'} 
{attribute 'no_explicit_call' := 'This FB is a CLASS and must be accessed using methods or properties'}
{attribute 'enable_dynamic_creation'}
FUNCTION_BLOCK _GVCP_REGISTER_ADDRESS EXTENDS AliasDatatypeBase
VAR
	localData : GVCP_REGISTER_ADDRESS;
	activeData : REFERENCE TO GVCP_REGISTER_ADDRESS REF= localData;
	aliasBaseDatatype : _UDINT(0);
END_VAR

PROPERTY PUBLIC Address : PVOID
GET
Address := ADR(activeData);
END_GET
END_PROPERTY

METHOD PUBLIC ClearReference
VAR_INPUT
END_VAR
activeData REF= localData;
SetBaseDatatypeReference();
END_METHOD

METHOD PUBLIC Clone : I_Datatype
VAR
    pClone : POINTER TO _GVCP_REGISTER_ADDRESS;
END_VAR
pClone := __NEW(_GVCP_REGISTER_ADDRESS(InitialValue := Value));
Clone := pClone^;
END_METHOD

METHOD FB_init : BOOL
VAR_INPUT
	bInitRetains : BOOL; // if TRUE, the retain variables are initialized (warm start / cold start)
	bInCopyCode : BOOL;  // if TRUE, the instance afterwards gets moved into the copy code (online change)
	InitialValue : GVCP_REGISTER_ADDRESS; // if possible, not all values can be initialized
END_VAR
localData := InitialValue;
SetBaseDatatypeReference();
AddBaseDatatype(aliasBaseDatatype);
END_METHOD

PROPERTY PUBLIC Identifier : T_MAXSTRING
GET
Identifier := 'GVCP_REGISTER_ADDRESS';
END_GET
END_PROPERTY

METHOD PUBLIC MakeReferenceTo
VAR_INPUT
	ReferenceTarget : REFERENCE TO GVCP_REGISTER_ADDRESS;
END_VAR
activeData REF= ReferenceTarget;
SetBaseDatatypeReference();
END_METHOD

METHOD PROTECTED SetBaseDatatypeReference
VAR_INPUT
END_VAR
aliasBaseDatatype.MakeReferenceTo(activeData);
END_METHOD

PROPERTY PUBLIC Size : UDINT
GET
Size := SIZEOF(activeData);
END_GET
END_PROPERTY

METHOD TryMakeReferenceTo : BOOL
VAR_INPUT
	Target : I_Datatype;
END_VAR
VAR
	pTargetData : POINTER TO GVCP_REGISTER_ADDRESS;
END_VAR
IF NOT IsEquivalentTo(Target) THEN
	RETURN;
END_IF

pTargetData := Target.Address;
activeData REF= pTargetData^;
SetBaseDatatypeReference();
TryMakeReferenceTo := TRUE;
END_METHOD

PROPERTY PUBLIC Value : REFERENCE TO GVCP_REGISTER_ADDRESS
GET
Value REF= activeData;
END_GET
END_PROPERTY

END_FUNCTION_BLOCK

// ---- Datatypes/Aliases/_TcVnMatrix2x3_LREAL.TcPOU
{attribute 'linkalways'} 
{attribute 'no_explicit_call' := 'This FB is a CLASS and must be accessed using methods or properties'}
{attribute 'enable_dynamic_creation'}
FUNCTION_BLOCK _TcVnMatrix2x3_LREAL EXTENDS AliasDatatypeBase
VAR
	localData : TcVnMatrix2x3_LREAL;
	activeData : REFERENCE TO TcVnMatrix2x3_LREAL REF= localData;
	aliasBaseDatatype : _Array0to1_0to2OfLREAL;
END_VAR

PROPERTY PUBLIC Address : PVOID
GET
Address := ADR(activeData);
END_GET
END_PROPERTY

METHOD PUBLIC ClearReference
VAR_INPUT
END_VAR
activeData REF= localData;
SetBaseDatatypeReference();
END_METHOD

METHOD PUBLIC Clone : I_Datatype
VAR
    pClone : POINTER TO _TcVnMatrix2x3_LREAL;
END_VAR
pClone := __NEW(_TcVnMatrix2x3_LREAL);
Clone := pClone^;
END_METHOD

METHOD FB_init : BOOL
VAR_INPUT
	bInitRetains : BOOL; // if TRUE, the retain variables are initialized (warm start / cold start)
	bInCopyCode : BOOL;  // if TRUE, the instance afterwards gets moved into the copy code (online change)
	//InitialValue : TcVnMatrix2x3_LREAL; // if possible, not all values can be initialized
END_VAR
//localData := InitialValue; // if possible, not all values can be initialized
SetBaseDatatypeReference();
AddBaseDatatype(aliasBaseDatatype);
END_METHOD

PROPERTY PUBLIC Identifier : T_MAXSTRING
GET
Identifier := 'TcVnMatrix2x3_LREAL';
END_GET
END_PROPERTY

METHOD PUBLIC MakeReferenceTo
VAR_INPUT
	ReferenceTarget : REFERENCE TO TcVnMatrix2x3_LREAL;
END_VAR
activeData REF= ReferenceTarget;
SetBaseDatatypeReference();
END_METHOD

METHOD PROTECTED SetBaseDatatypeReference
VAR_INPUT
END_VAR
aliasBaseDatatype.MakeReferenceTo(activeData);
END_METHOD

PROPERTY PUBLIC Size : UDINT
GET
Size := SIZEOF(activeData);
END_GET
END_PROPERTY

METHOD TryMakeReferenceTo : BOOL
VAR_INPUT
	Target : I_Datatype;
END_VAR
VAR
	pTargetData : POINTER TO TcVnMatrix2x3_LREAL;
END_VAR
IF NOT IsEquivalentTo(Target) THEN
	RETURN;
END_IF

pTargetData := Target.Address;
activeData REF= pTargetData^;
SetBaseDatatypeReference();
TryMakeReferenceTo := TRUE;
END_METHOD

PROPERTY PUBLIC Value : REFERENCE TO TcVnMatrix2x3_LREAL
GET
Value REF= activeData;
END_GET
END_PROPERTY

END_FUNCTION_BLOCK

// ---- Datatypes/Arrays/_Array0to1_0to2OfLREAL.TcPOU
{attribute 'linkalways'} 
{attribute 'no_explicit_call' := 'This FB is a CLASS and must be accessed using methods or properties'}
{attribute 'enable_dynamic_creation'}
FUNCTION_BLOCK _Array0to1_0to2OfLREAL EXTENDS ArrayDatatypeBase_2D
VAR CONSTANT
	lBoundD1 : DINT := 0;
	uBoundD1 : DINT := 1;
	lBoundD2 : DINT := 0;
	uBoundD2 : DINT := 2;
END_VAR
VAR
	localData : ARRAY [lBoundD1..uBoundD1,lBoundD2..uBoundD2] OF LREAL;
	activeData : REFERENCE TO ARRAY [lBoundD1..uBoundD1,lBoundD2..uBoundD2] OF LREAL REF= localData;
	elements : ARRAY [lBoundD1..uBoundD1,lBoundD2..uBoundD2] OF _LREAL(0);
	baseType : _LREAL(0);
END_VAR

PROPERTY PUBLIC Address : PVOID
GET
Address := ADR(activeData);
END_GET
END_PROPERTY

PROPERTY PUBLIC BaseDatatype : I_Datatype
GET
BaseDatatype := baseType;
END_GET
END_PROPERTY

METHOD PUBLIC ClearReference
VAR_INPUT
END_VAR
activeData REF= localData;
SetElementReference();
END_METHOD

METHOD PUBLIC Clone : I_Datatype
VAR
    pClone : POINTER TO _Array0to1_0to2OfLREAL;
END_VAR
pClone := __NEW(_Array0to1_0to2OfLREAL());
pClone^.Value := Value;
Clone := pClone^;
END_METHOD

METHOD FB_init : BOOL
VAR_INPUT
	bInitRetains : BOOL; // if TRUE, the retain variables are initialized (warm start / cold start)
	bInCopyCode : BOOL;  // if TRUE, the instance afterwards gets moved into the copy code (online change)
END_VAR
SetElementReference();
END_METHOD

METHOD PUBLIC MakeReferenceTo
VAR_INPUT
	ReferenceTarget : REFERENCE TO ARRAY [lBoundD1..uBoundD1,lBoundD2..uBoundD2] OF LREAL;
END_VAR
activeData REF= ReferenceTarget;
SetElementReference();
END_METHOD

METHOD PROTECTED OnSerializeArrayValues
VAR_INPUT
	Serializer : I_Serializer;
END_VAR
VAR
	i, j : DINT;
END_VAR
FOR i := lBoundD1 TO uBoundD1 DO
	Serializer.StartArray();
	FOR j := lBoundD2 TO uBoundD2 DO
		elements[i, j].SerializeWith(Serializer);
	END_FOR
	Serializer.EndArray();
END_FOR
END_METHOD

METHOD PROTECTED SetElementReference
VAR_INPUT
END_VAR
VAR
	i, j : DINT;
END_VAR
FOR i := lBoundD1 TO uBoundD1 DO
	FOR j := lBoundD2 TO uBoundD2 DO
		elements[i, j].MakeReferenceTo(activeData[i, j]);
	END_FOR
END_FOR
END_METHOD

PROPERTY PUBLIC Size : UDINT
GET
Size := SIZEOF(activeData);
END_GET
END_PROPERTY

METHOD PROTECTED TryDeserializeArrayValues : BOOL
VAR_INPUT
	Deserializer : I_Deserializer;
	Feedback : I_DeserializerFeedback;
END_VAR
VAR
	enumeratorD1 : I_DeserializerArrayForwardEnumerator;
	enumeratorD2 : I_DeserializerArrayForwardEnumerator;
	i, j : DINT;
END_VAR
enumeratorD1 := Deserializer.GetArrayEnumerator();
i := lBoundD1;

WHILE enumeratorD1.MoveNext() AND i <= uBoundD1 DO
	
	enumeratorD2 := enumeratorD1.Current.GetArrayEnumerator();
	j := lBoundD2;
	
	WHILE enumeratorD2.MoveNext() AND j <= uBoundD2 DO
	
		IF NOT elements[i, j].TryDeserializeFrom(enumeratorD2.Current, Feedback) THEN
			EXIT;
		END_IF
		
		j := j + 1;
	
	END_WHILE
	enumeratorD2.Dispose();

	i := i + 1;

END_WHILE
enumeratorD1.Dispose();
END_METHOD

METHOD PUBLIC TryGetElementAsDatatypeByIndex : BOOL
VAR_INPUT
	Index1 : DINT;
	Index2 : DINT;
	Destination : REFERENCE TO I_Datatype;
END_VAR
IF Index1 < lboundD1 OR Index1 > uboundD1 THEN
	RETURN;
END_IF

IF Index2 < lboundD2 OR Index2 > uboundD2 THEN
	RETURN;
END_IF

Destination := elements[Index1, Index2];
TryGetElementAsDatatypeByIndex := TRUE;
END_METHOD

METHOD PUBLIC TryGetLowerBound : BOOL
VAR_INPUT
	Dimention : UDINT;
	Destination : REFERENCE TO DINT;
END_VAR
CASE Dimention OF
	
	1:	Destination := lBoundD1;
		TryGetLowerBound := TRUE;
		RETURN;
	
	2:	Destination := lBoundD2;
		TryGetLowerBound := TRUE;
		RETURN;

END_CASE
END_METHOD

METHOD PUBLIC TryGetUpperBound : BOOL
VAR_INPUT
	Dimention : UDINT;
	Destination : REFERENCE TO DINT;
END_VAR
CASE Dimention OF
	
	1:	Destination := uBoundD1;
		TryGetUpperBound := TRUE;
		RETURN;
	
	2:	Destination := uBoundD2;
		TryGetUpperBound := TRUE;
		RETURN;

END_CASE
END_METHOD

METHOD TryMakeReferenceTo : BOOL
VAR_INPUT
	Target : I_Datatype;
END_VAR
VAR
	pTargetData : POINTER TO ARRAY [lBoundD1..uBoundD1,lBoundD2..uBoundD2] OF LREAL;
END_VAR
IF NOT IsEquivalentTo(Target) THEN
	RETURN;
END_IF

pTargetData := Target.Address;
activeData REF= pTargetData^;
SetElementReference();
TryMakeReferenceTo := TRUE;
END_METHOD

PROPERTY PUBLIC Value : REFERENCE TO ARRAY [lBoundD1..uBoundD1,lBoundD2..uBoundD2] OF LREAL;
GET
Value ref= activeData;
END_GET
END_PROPERTY

END_FUNCTION_BLOCK

// ---- Datatypes/Aliases/_TcVnArray7_LREAL.TcPOU
{attribute 'linkalways'} 
{attribute 'no_explicit_call' := 'This FB is a CLASS and must be accessed using methods or properties'}
{attribute 'enable_dynamic_creation'}
FUNCTION_BLOCK _TcVnArray7_LREAL EXTENDS AliasDatatypeBase
VAR
	localData : TcVnArray7_LREAL;
	activeData : REFERENCE TO TcVnArray7_LREAL REF= localData;
	aliasBaseDatatype : _Array0to6OfLREAL;
END_VAR

PROPERTY PUBLIC Address : PVOID
GET
Address := ADR(activeData);
END_GET
END_PROPERTY

METHOD PUBLIC ClearReference
VAR_INPUT
END_VAR
activeData REF= localData;
SetBaseDatatypeReference();
END_METHOD

METHOD PUBLIC Clone : I_Datatype
VAR
    pClone : POINTER TO _TcVnArray7_LREAL;
END_VAR
pClone := __NEW(_TcVnArray7_LREAL);
Clone := pClone^;
END_METHOD

METHOD FB_init : BOOL
VAR_INPUT
	bInitRetains : BOOL; // if TRUE, the retain variables are initialized (warm start / cold start)
	bInCopyCode : BOOL;  // if TRUE, the instance afterwards gets moved into the copy code (online change)
	//InitialValue : TcVnArray7_LREAL; // if possible, not all values can be initialized
END_VAR
//localData := InitialValue; // if possible, not all values can be initialized
SetBaseDatatypeReference();
AddBaseDatatype(aliasBaseDatatype);
END_METHOD

PROPERTY PUBLIC Identifier : T_MAXSTRING
GET
Identifier := 'TcVnArray7_LREAL';
END_GET
END_PROPERTY

METHOD PUBLIC MakeReferenceTo
VAR_INPUT
	ReferenceTarget : REFERENCE TO TcVnArray7_LREAL;
END_VAR
activeData REF= ReferenceTarget;
SetBaseDatatypeReference();
END_METHOD

METHOD PROTECTED SetBaseDatatypeReference
VAR_INPUT
END_VAR
aliasBaseDatatype.MakeReferenceTo(activeData);
END_METHOD

PROPERTY PUBLIC Size : UDINT
GET
Size := SIZEOF(activeData);
END_GET
END_PROPERTY

METHOD TryMakeReferenceTo : BOOL
VAR_INPUT
	Target : I_Datatype;
END_VAR
VAR
	pTargetData : POINTER TO TcVnArray7_LREAL;
END_VAR
IF NOT IsEquivalentTo(Target) THEN
	RETURN;
END_IF

pTargetData := Target.Address;
activeData REF= pTargetData^;
SetBaseDatatypeReference();
TryMakeReferenceTo := TRUE;
END_METHOD

PROPERTY PUBLIC Value : REFERENCE TO TcVnArray7_LREAL
GET
Value REF= activeData;
END_GET
END_PROPERTY

END_FUNCTION_BLOCK

// ---- Datatypes/Aliases/_TcVnArray8_LREAL.TcPOU
{attribute 'linkalways'} 
{attribute 'no_explicit_call' := 'This FB is a CLASS and must be accessed using methods or properties'}
{attribute 'enable_dynamic_creation'}
FUNCTION_BLOCK _TcVnArray8_LREAL EXTENDS AliasDatatypeBase
VAR
	localData : TcVnArray8_LREAL;
	activeData : REFERENCE TO TcVnArray8_LREAL REF= localData;
	aliasBaseDatatype : _Array0to7OfLREAL;
END_VAR

PROPERTY PUBLIC Address : PVOID
GET
Address := ADR(activeData);
END_GET
END_PROPERTY

METHOD PUBLIC ClearReference
VAR_INPUT
END_VAR
activeData REF= localData;
SetBaseDatatypeReference();
END_METHOD

METHOD PUBLIC Clone : I_Datatype
VAR
    pClone : POINTER TO _TcVnArray8_LREAL;
END_VAR
pClone := __NEW(_TcVnArray8_LREAL);
Clone := pClone^;
END_METHOD

METHOD FB_init : BOOL
VAR_INPUT
	bInitRetains : BOOL; // if TRUE, the retain variables are initialized (warm start / cold start)
	bInCopyCode : BOOL;  // if TRUE, the instance afterwards gets moved into the copy code (online change)
	//InitialValue : TcVnArray8_LREAL; // if possible, not all values can be initialized
END_VAR
//localData := InitialValue; // if possible, not all values can be initialized
SetBaseDatatypeReference();
AddBaseDatatype(aliasBaseDatatype);
END_METHOD

PROPERTY PUBLIC Identifier : T_MAXSTRING
GET
Identifier := 'TcVnArray8_LREAL';
END_GET
END_PROPERTY

METHOD PUBLIC MakeReferenceTo
VAR_INPUT
	ReferenceTarget : REFERENCE TO TcVnArray8_LREAL;
END_VAR
activeData REF= ReferenceTarget;
SetBaseDatatypeReference();
END_METHOD

METHOD PROTECTED SetBaseDatatypeReference
VAR_INPUT
END_VAR
aliasBaseDatatype.MakeReferenceTo(activeData);
END_METHOD

PROPERTY PUBLIC Size : UDINT
GET
Size := SIZEOF(activeData);
END_GET
END_PROPERTY

METHOD TryMakeReferenceTo : BOOL
VAR_INPUT
	Target : I_Datatype;
END_VAR
VAR
	pTargetData : POINTER TO TcVnArray8_LREAL;
END_VAR
IF NOT IsEquivalentTo(Target) THEN
	RETURN;
END_IF

pTargetData := Target.Address;
activeData REF= pTargetData^;
SetBaseDatatypeReference();
TryMakeReferenceTo := TRUE;
END_METHOD

PROPERTY PUBLIC Value : REFERENCE TO TcVnArray8_LREAL
GET
Value REF= activeData;
END_GET
END_PROPERTY

END_FUNCTION_BLOCK

// ---- Datatypes/Arrays/_Array0to7OfLREAL.TcPOU
{attribute 'linkalways'} 
{attribute 'no_explicit_call' := 'This FB is a CLASS and must be accessed using methods or properties'}
{attribute 'enable_dynamic_creation'}
FUNCTION_BLOCK _Array0to7OfLREAL EXTENDS ArrayDatatypeBase_1D
VAR CONSTANT
	lBound : DINT := 0;
	uBound : DINT := 7;
END_VAR
VAR
	localData : ARRAY [lBound..uBound] OF LREAL;
	activeData : REFERENCE TO ARRAY [lBound..uBound] OF LREAL REF= localData;
	elements : ARRAY [lBound..uBound] OF _LREAL(0.0);
	baseType : _LREAL(0.0);
END_VAR

PROPERTY PUBLIC Address : PVOID
GET
Address := ADR(activeData);
END_GET
END_PROPERTY

PROPERTY PUBLIC BaseDatatype : I_Datatype
GET
BaseDatatype := baseType;
END_GET
END_PROPERTY

METHOD PUBLIC ClearReference
VAR_INPUT
END_VAR
activeData REF= localData;
SetElementReference();
END_METHOD

METHOD PUBLIC Clone : I_Datatype
VAR
    pClone : POINTER TO _Array0to7OfLREAL;
END_VAR
pClone := __NEW(_Array0to7OfLREAL());
pClone^.Value := Value;
Clone := pClone^;
END_METHOD

METHOD FB_init : BOOL
VAR_INPUT
	bInitRetains : BOOL; // if TRUE, the retain variables are initialized (warm start / cold start)
	bInCopyCode : BOOL;  // if TRUE, the instance afterwards gets moved into the copy code (online change)
END_VAR
SetElementReference();
END_METHOD

METHOD PUBLIC MakeReferenceTo
VAR_INPUT
	ReferenceTarget : REFERENCE TO ARRAY [lBound..uBound] OF LREAL;
END_VAR
activeData REF= ReferenceTarget;
SetElementReference();
END_METHOD

METHOD PROTECTED OnSerializeArrayValues
VAR_INPUT
	Serializer : I_Serializer;
END_VAR
VAR
	i : DINT;
END_VAR
FOR i := lBound TO uBound DO
	elements[i].SerializeWith(Serializer);
END_FOR
END_METHOD

METHOD PROTECTED SetElementReference
VAR_INPUT
END_VAR
VAR
	i : DINT;
END_VAR
FOR i := lBound TO uBound DO
	elements[i].MakeReferenceTo(activeData[i]);
END_FOR
END_METHOD

PROPERTY PUBLIC Size : UDINT
GET
Size := SIZEOF(activeData);
END_GET
END_PROPERTY

METHOD PROTECTED TryDeserializeArrayValues : BOOL
VAR_INPUT
	Deserializer : I_Deserializer;
	Feedback : I_DeserializerFeedback;
END_VAR
VAR
	enumerator : I_DeserializerArrayForwardEnumerator;
	i : DINT;
END_VAR
enumerator := Deserializer.GetArrayEnumerator();
i := lBound;

WHILE enumerator.MoveNext() AND i <= uBound DO
	
	IF NOT elements[i].TryDeserializeFrom(enumerator.Current, Feedback) THEN
		EXIT;
	END_IF
	i := i + 1;

END_WHILE
enumerator.Dispose();
END_METHOD

METHOD PUBLIC TryGetElementAsDatatypeByIndex : BOOL
VAR_INPUT
	Index : DINT;
	Destination : REFERENCE TO I_Datatype;
END_VAR
IF Index < lbound OR Index > ubound THEN
	RETURN;
END_IF

Destination := elements[Index];
TryGetElementAsDatatypeByIndex := TRUE;
END_METHOD

METHOD PUBLIC TryGetLowerBound : BOOL
VAR_INPUT
	Dimention : UDINT;
	Destination : REFERENCE TO DINT;
END_VAR
IF Dimention = 1 THEN
	Destination := lBound;
	TryGetLowerBound := TRUE;
END_IF
END_METHOD

METHOD PUBLIC TryGetUpperBound : BOOL
VAR_INPUT
	Dimention : UDINT;
	Destination : REFERENCE TO DINT;
END_VAR
IF Dimention = 1 THEN
	Destination := uBound;
	TryGetUpperBound := TRUE;
END_IF
END_METHOD

METHOD TryMakeReferenceTo : BOOL
VAR_INPUT
	Target : I_Datatype;
END_VAR
VAR
	pTargetData : POINTER TO ARRAY [lBound..uBound] OF LREAL;
END_VAR
IF NOT IsEquivalentTo(Target) THEN
	RETURN;
END_IF

pTargetData := Target.Address;
activeData REF= pTargetData^;
SetElementReference();
TryMakeReferenceTo := TRUE;
END_METHOD

PROPERTY PUBLIC Value : REFERENCE TO ARRAY [lBound..uBound] OF LREAL;
GET
Value ref= activeData;
END_GET
END_PROPERTY

END_FUNCTION_BLOCK

// ---- Datatypes/Aliases/_TcVnPoint3_REAL.TcPOU
{attribute 'linkalways'} 
{attribute 'no_explicit_call' := 'This FB is a CLASS and must be accessed using methods or properties'}
{attribute 'enable_dynamic_creation'}
FUNCTION_BLOCK _TcVnPoint3_REAL EXTENDS AliasDatatypeBase
VAR
	localData : TcVnPoint3_REAL;
	activeData : REFERENCE TO TcVnPoint3_REAL REF= localData;
	aliasBaseDatatype : _TcVnVector3_REAL;
END_VAR

PROPERTY PUBLIC Address : PVOID
GET
Address := ADR(activeData);
END_GET
END_PROPERTY

METHOD PUBLIC ClearReference
VAR_INPUT
END_VAR
activeData REF= localData;
SetBaseDatatypeReference();
END_METHOD

METHOD PUBLIC Clone : I_Datatype
VAR
    pClone : POINTER TO _TcVnPoint3_REAL;
END_VAR
pClone := __NEW(_TcVnPoint3_REAL);
Clone := pClone^;
END_METHOD

METHOD FB_init : BOOL
VAR_INPUT
	bInitRetains : BOOL; // if TRUE, the retain variables are initialized (warm start / cold start)
	bInCopyCode : BOOL;  // if TRUE, the instance afterwards gets moved into the copy code (online change)
	//InitialValue : <type>; // if possible, not all values can be initialized
END_VAR
//localData := InitialValue; // if possible, not all values can be initialized
SetBaseDatatypeReference();
AddBaseDatatype(aliasBaseDatatype);
END_METHOD

PROPERTY PUBLIC Identifier : T_MAXSTRING
GET
Identifier := 'TcVnPoint3_REAL';
END_GET
END_PROPERTY

METHOD PUBLIC MakeReferenceTo
VAR_INPUT
	ReferenceTarget : REFERENCE TO TcVnPoint3_REAL;
END_VAR
activeData REF= ReferenceTarget;
SetBaseDatatypeReference();
END_METHOD

METHOD PROTECTED SetBaseDatatypeReference
VAR_INPUT
END_VAR
aliasBaseDatatype.MakeReferenceTo(activeData);
END_METHOD

PROPERTY PUBLIC Size : UDINT
GET
Size := SIZEOF(activeData);
END_GET
END_PROPERTY

METHOD TryMakeReferenceTo : BOOL
VAR_INPUT
	Target : I_Datatype;
END_VAR
VAR
	pTargetData : POINTER TO TcVnPoint3_REAL;
END_VAR
IF NOT IsEquivalentTo(Target) THEN
	RETURN;
END_IF

pTargetData := Target.Address;
activeData REF= pTargetData^;
SetBaseDatatypeReference();
TryMakeReferenceTo := TRUE;
END_METHOD

PROPERTY PUBLIC Value : REFERENCE TO TcVnPoint3_REAL
GET
Value REF= activeData;
END_GET
END_PROPERTY

END_FUNCTION_BLOCK

// ---- Datatypes/Aliases/_TcVnVector3_REAL.TcPOU
{attribute 'linkalways'} 
{attribute 'no_explicit_call' := 'This FB is a CLASS and must be accessed using methods or properties'}
{attribute 'enable_dynamic_creation'}
FUNCTION_BLOCK _TcVnVector3_REAL EXTENDS AliasDatatypeBase
VAR
	localData : TcVnVector3_REAL;
	activeData : REFERENCE TO TcVnVector3_REAL REF= localData;
	aliasBaseDatatype : _Array0to2OfREAL;
END_VAR

PROPERTY PUBLIC Address : PVOID
GET
Address := ADR(activeData);
END_GET
END_PROPERTY

METHOD PUBLIC ClearReference
VAR_INPUT
END_VAR
activeData REF= localData;
SetBaseDatatypeReference();
END_METHOD

METHOD PUBLIC Clone : I_Datatype
VAR
    pClone : POINTER TO _TcVnVector3_REAL;
END_VAR
pClone := __NEW(_TcVnVector3_REAL);
Clone := pClone^;
END_METHOD

METHOD FB_init : BOOL
VAR_INPUT
	bInitRetains : BOOL; // if TRUE, the retain variables are initialized (warm start / cold start)
	bInCopyCode : BOOL;  // if TRUE, the instance afterwards gets moved into the copy code (online change)
	//InitialValue : <type>; // if possible, not all values can be initialized
END_VAR
//localData := InitialValue; // if possible, not all values can be initialized
SetBaseDatatypeReference();
AddBaseDatatype(aliasBaseDatatype);
END_METHOD

PROPERTY PUBLIC Identifier : T_MAXSTRING
GET
Identifier := 'TcVnVector3_REAL';
END_GET
END_PROPERTY

METHOD PUBLIC MakeReferenceTo
VAR_INPUT
	ReferenceTarget : REFERENCE TO TcVnVector3_REAL;
END_VAR
activeData REF= ReferenceTarget;
SetBaseDatatypeReference();
END_METHOD

METHOD PROTECTED SetBaseDatatypeReference
VAR_INPUT
END_VAR
aliasBaseDatatype.MakeReferenceTo(activeData);
END_METHOD

PROPERTY PUBLIC Size : UDINT
GET
Size := SIZEOF(activeData);
END_GET
END_PROPERTY

METHOD TryMakeReferenceTo : BOOL
VAR_INPUT
	Target : I_Datatype;
END_VAR
VAR
	pTargetData : POINTER TO TcVnVector3_REAL;
END_VAR
IF NOT IsEquivalentTo(Target) THEN
	RETURN;
END_IF

pTargetData := Target.Address;
activeData REF= pTargetData^;
SetBaseDatatypeReference();
TryMakeReferenceTo := TRUE;
END_METHOD

PROPERTY PUBLIC Value : REFERENCE TO TcVnVector3_REAL
GET
Value REF= activeData;
END_GET
END_PROPERTY

END_FUNCTION_BLOCK

// ---- Datatypes/Arrays/_Array0to2OfREAL.TcPOU
{attribute 'linkalways'} 
{attribute 'no_explicit_call' := 'This FB is a CLASS and must be accessed using methods or properties'}
{attribute 'enable_dynamic_creation'}
FUNCTION_BLOCK _Array0to2OfREAL EXTENDS ArrayDatatypeBase_1D
VAR CONSTANT
	lBound : DINT := 0;
	uBound : DINT := 2;
END_VAR
VAR
	localData : ARRAY [lBound..uBound] OF REAL;
	activeData : REFERENCE TO ARRAY [lBound..uBound] OF REAL REF= localData;
	elements : ARRAY [lBound..uBound] OF _REAL(0.0);
	baseType : _REAL(0.0);
END_VAR

PROPERTY PUBLIC Address : PVOID
GET
Address := ADR(activeData);
END_GET
END_PROPERTY

PROPERTY PUBLIC BaseDatatype : I_Datatype
GET
BaseDatatype := baseType;
END_GET
END_PROPERTY

METHOD PUBLIC ClearReference
VAR_INPUT
END_VAR
activeData REF= localData;
SetElementReference();
END_METHOD

METHOD PUBLIC Clone : I_Datatype
VAR
    pClone : POINTER TO _Array0to2OfREAL;
END_VAR
pClone := __NEW(_Array0to2OfREAL());
pClone^.Value := Value;
Clone := pClone^;
END_METHOD

METHOD FB_init : BOOL
VAR_INPUT
	bInitRetains : BOOL; // if TRUE, the retain variables are initialized (warm start / cold start)
	bInCopyCode : BOOL;  // if TRUE, the instance afterwards gets moved into the copy code (online change)
END_VAR
SetElementReference();
END_METHOD

METHOD PUBLIC MakeReferenceTo
VAR_INPUT
	ReferenceTarget : REFERENCE TO ARRAY [lBound..uBound] OF REAL;
END_VAR
activeData REF= ReferenceTarget;
SetElementReference();
END_METHOD

METHOD PROTECTED OnSerializeArrayValues
VAR_INPUT
	Serializer : I_Serializer;
END_VAR
VAR
	i : DINT;
END_VAR
FOR i := lBound TO uBound DO
	elements[i].SerializeWith(Serializer);
END_FOR
END_METHOD

METHOD PROTECTED SetElementReference
VAR_INPUT
END_VAR
VAR
	i : DINT;
END_VAR
FOR i := lBound TO uBound DO
	elements[i].MakeReferenceTo(activeData[i]);
END_FOR
END_METHOD

PROPERTY PUBLIC Size : UDINT
GET
Size := SIZEOF(activeData);
END_GET
END_PROPERTY

METHOD PROTECTED TryDeserializeArrayValues : BOOL
VAR_INPUT
	Deserializer : I_Deserializer;
	Feedback : I_DeserializerFeedback;
END_VAR
VAR
	enumerator : I_DeserializerArrayForwardEnumerator;
	i : DINT;
END_VAR
enumerator := Deserializer.GetArrayEnumerator();
i := lBound;

WHILE enumerator.MoveNext() AND i <= uBound DO
	
	IF NOT elements[i].TryDeserializeFrom(enumerator.Current, Feedback) THEN
		EXIT;
	END_IF
	i := i + 1;

END_WHILE
enumerator.Dispose();
END_METHOD

METHOD PUBLIC TryGetElementAsDatatypeByIndex : BOOL
VAR_INPUT
	Index : DINT;
	Destination : REFERENCE TO I_Datatype;
END_VAR
IF Index < lbound OR Index > ubound THEN
	RETURN;
END_IF

Destination := elements[Index];
TryGetElementAsDatatypeByIndex := TRUE;
END_METHOD

METHOD PUBLIC TryGetLowerBound : BOOL
VAR_INPUT
	Dimention : UDINT;
	Destination : REFERENCE TO DINT;
END_VAR
IF Dimention = 1 THEN
	Destination := lBound;
	TryGetLowerBound := TRUE;
END_IF
END_METHOD

METHOD PUBLIC TryGetUpperBound : BOOL
VAR_INPUT
	Dimention : UDINT;
	Destination : REFERENCE TO DINT;
END_VAR
IF Dimention = 1 THEN
	Destination := uBound;
	TryGetUpperBound := TRUE;
END_IF
END_METHOD

METHOD TryMakeReferenceTo : BOOL
VAR_INPUT
	Target : I_Datatype;
END_VAR
VAR
	pTargetData : POINTER TO ARRAY [lBound..uBound] OF REAL;
END_VAR
IF NOT IsEquivalentTo(Target) THEN
	RETURN;
END_IF

pTargetData := Target.Address;
activeData REF= pTargetData^;
SetElementReference();
TryMakeReferenceTo := TRUE;
END_METHOD

PROPERTY PUBLIC Value : REFERENCE TO ARRAY [lBound..uBound] OF REAL;
GET
Value ref= activeData;
END_GET
END_PROPERTY

END_FUNCTION_BLOCK

// ---- Datatypes/Aliases/_TcVnPoint3_LREAL.TcPOU
{attribute 'linkalways'} 
{attribute 'no_explicit_call' := 'This FB is a CLASS and must be accessed using methods or properties'}
{attribute 'enable_dynamic_creation'}
FUNCTION_BLOCK _TcVnPoint3_LREAL EXTENDS AliasDatatypeBase
VAR
	localData : TcVnPoint3_LREAL;
	activeData : REFERENCE TO TcVnPoint3_LREAL REF= localData;
	aliasBaseDatatype : _TcVnVector3_LREAL;
END_VAR

PROPERTY PUBLIC Address : PVOID
GET
Address := ADR(activeData);
END_GET
END_PROPERTY

METHOD PUBLIC ClearReference
VAR_INPUT
END_VAR
activeData REF= localData;
SetBaseDatatypeReference();
END_METHOD

METHOD PUBLIC Clone : I_Datatype
VAR
    pClone : POINTER TO _TcVnPoint3_LREAL;
END_VAR
pClone := __NEW(_TcVnPoint3_LREAL);
Clone := pClone^;
END_METHOD

METHOD FB_init : BOOL
VAR_INPUT
	bInitRetains : BOOL; // if TRUE, the retain variables are initialized (warm start / cold start)
	bInCopyCode : BOOL;  // if TRUE, the instance afterwards gets moved into the copy code (online change)
	//InitialValue : <type>; // if possible, not all values can be initialized
END_VAR
//localData := InitialValue; // if possible, not all values can be initialized
SetBaseDatatypeReference();
AddBaseDatatype(aliasBaseDatatype);
END_METHOD

PROPERTY PUBLIC Identifier : T_MAXSTRING
GET
Identifier := 'TcVnPoint3_LREAL';
END_GET
END_PROPERTY

METHOD PUBLIC MakeReferenceTo
VAR_INPUT
	ReferenceTarget : REFERENCE TO TcVnPoint3_LREAL;
END_VAR
activeData REF= ReferenceTarget;
SetBaseDatatypeReference();
END_METHOD

METHOD PROTECTED SetBaseDatatypeReference
VAR_INPUT
END_VAR
aliasBaseDatatype.MakeReferenceTo(activeData);
END_METHOD

PROPERTY PUBLIC Size : UDINT
GET
Size := SIZEOF(activeData);
END_GET
END_PROPERTY

METHOD TryMakeReferenceTo : BOOL
VAR_INPUT
	Target : I_Datatype;
END_VAR
VAR
	pTargetData : POINTER TO TcVnPoint3_LREAL;
END_VAR
IF NOT IsEquivalentTo(Target) THEN
	RETURN;
END_IF

pTargetData := Target.Address;
activeData REF= pTargetData^;
SetBaseDatatypeReference();
TryMakeReferenceTo := TRUE;
END_METHOD

PROPERTY PUBLIC Value : REFERENCE TO TcVnPoint3_LREAL
GET
Value REF= activeData;
END_GET
END_PROPERTY

END_FUNCTION_BLOCK

// ---- Datatypes/Aliases/_TcVnVector2_DINT.TcPOU
{attribute 'linkalways'} 
{attribute 'no_explicit_call' := 'This FB is a CLASS and must be accessed using methods or properties'}
{attribute 'enable_dynamic_creation'}
FUNCTION_BLOCK _TcVnVector2_DINT EXTENDS AliasDatatypeBase
VAR
	localData : TcVnVector2_DINT;
	activeData : REFERENCE TO TcVnVector2_DINT REF= localData;
	aliasBaseDatatype : _Array0to1OfDINT;
END_VAR

PROPERTY PUBLIC Address : PVOID
GET
Address := ADR(activeData);
END_GET
END_PROPERTY

METHOD PUBLIC ClearReference
VAR_INPUT
END_VAR
activeData REF= localData;
SetBaseDatatypeReference();
END_METHOD

METHOD PUBLIC Clone : I_Datatype
VAR
    pClone : POINTER TO _TcVnVector2_DINT;
END_VAR
pClone := __NEW(_TcVnVector2_DINT);
Clone := pClone^;
END_METHOD

METHOD FB_init : BOOL
VAR_INPUT
	bInitRetains : BOOL; // if TRUE, the retain variables are initialized (warm start / cold start)
	bInCopyCode : BOOL;  // if TRUE, the instance afterwards gets moved into the copy code (online change)
	//InitialValue : <type>; // if possible, not all values can be initialized
END_VAR
//localData := InitialValue; // if possible, not all values can be initialized
SetBaseDatatypeReference();
AddBaseDatatype(aliasBaseDatatype);
END_METHOD

PROPERTY PUBLIC Identifier : T_MAXSTRING
GET
Identifier := 'TcVnVector2_DINT';
END_GET
END_PROPERTY

METHOD PUBLIC MakeReferenceTo
VAR_INPUT
	ReferenceTarget : REFERENCE TO TcVnVector2_DINT;
END_VAR
activeData REF= ReferenceTarget;
SetBaseDatatypeReference();
END_METHOD

METHOD PROTECTED SetBaseDatatypeReference
VAR_INPUT
END_VAR
aliasBaseDatatype.MakeReferenceTo(activeData);
END_METHOD

PROPERTY PUBLIC Size : UDINT
GET
Size := SIZEOF(activeData);
END_GET
END_PROPERTY

METHOD TryMakeReferenceTo : BOOL
VAR_INPUT
	Target : I_Datatype;
END_VAR
VAR
	pTargetData : POINTER TO TcVnVector2_DINT;
END_VAR
IF NOT IsEquivalentTo(Target) THEN
	RETURN;
END_IF

pTargetData := Target.Address;
activeData REF= pTargetData^;
SetBaseDatatypeReference();
TryMakeReferenceTo := TRUE;
END_METHOD

PROPERTY PUBLIC Value : REFERENCE TO TcVnVector2_DINT
GET
Value REF= activeData;
END_GET
END_PROPERTY

END_FUNCTION_BLOCK

// ---- Datatypes/Aliases/_TcVnVector3_INT.TcPOU
{attribute 'linkalways'} 
{attribute 'no_explicit_call' := 'This FB is a CLASS and must be accessed using methods or properties'}
{attribute 'enable_dynamic_creation'}
FUNCTION_BLOCK _TcVnVector3_INT EXTENDS AliasDatatypeBase
VAR
	localData : TcVnVector3_INT;
	activeData : REFERENCE TO TcVnVector3_INT REF= localData;
	aliasBaseDatatype : _Array0to2OfINT;
END_VAR

PROPERTY PUBLIC Address : PVOID
GET
Address := ADR(activeData);
END_GET
END_PROPERTY

METHOD PUBLIC ClearReference
VAR_INPUT
END_VAR
activeData REF= localData;
SetBaseDatatypeReference();
END_METHOD

METHOD PUBLIC Clone : I_Datatype
VAR
    pClone : POINTER TO _TcVnVector3_INT;
END_VAR
pClone := __NEW(_TcVnVector3_INT);
Clone := pClone^;
END_METHOD

METHOD FB_init : BOOL
VAR_INPUT
	bInitRetains : BOOL; // if TRUE, the retain variables are initialized (warm start / cold start)
	bInCopyCode : BOOL;  // if TRUE, the instance afterwards gets moved into the copy code (online change)
	//InitialValue : <type>; // if possible, not all values can be initialized
END_VAR
//localData := InitialValue; // if possible, not all values can be initialized
SetBaseDatatypeReference();
AddBaseDatatype(aliasBaseDatatype);
END_METHOD

PROPERTY PUBLIC Identifier : T_MAXSTRING
GET
Identifier := 'TcVnVector3_INT';
END_GET
END_PROPERTY

METHOD PUBLIC MakeReferenceTo
VAR_INPUT
	ReferenceTarget : REFERENCE TO TcVnVector3_INT;
END_VAR
activeData REF= ReferenceTarget;
SetBaseDatatypeReference();
END_METHOD

METHOD PROTECTED SetBaseDatatypeReference
VAR_INPUT
END_VAR
aliasBaseDatatype.MakeReferenceTo(activeData);
END_METHOD

PROPERTY PUBLIC Size : UDINT
GET
Size := SIZEOF(activeData);
END_GET
END_PROPERTY

METHOD TryMakeReferenceTo : BOOL
VAR_INPUT
	Target : I_Datatype;
END_VAR
VAR
	pTargetData : POINTER TO TcVnVector3_INT;
END_VAR
IF NOT IsEquivalentTo(Target) THEN
	RETURN;
END_IF

pTargetData := Target.Address;
activeData REF= pTargetData^;
SetBaseDatatypeReference();
TryMakeReferenceTo := TRUE;
END_METHOD

PROPERTY PUBLIC Value : REFERENCE TO TcVnVector3_INT
GET
Value REF= activeData;
END_GET
END_PROPERTY

END_FUNCTION_BLOCK

// ---- Datatypes/Aliases/_TcVnVector2_USINT.TcPOU
{attribute 'linkalways'} 
{attribute 'no_explicit_call' := 'This FB is a CLASS and must be accessed using methods or properties'}
{attribute 'enable_dynamic_creation'}
FUNCTION_BLOCK _TcVnVector2_USINT EXTENDS AliasDatatypeBase
VAR
	localData : TcVnVector2_USINT;
	activeData : REFERENCE TO TcVnVector2_USINT REF= localData;
	aliasBaseDatatype : _Array0to1OfUSINT;
END_VAR

PROPERTY PUBLIC Address : PVOID
GET
Address := ADR(activeData);
END_GET
END_PROPERTY

METHOD PUBLIC ClearReference
VAR_INPUT
END_VAR
activeData REF= localData;
SetBaseDatatypeReference();
END_METHOD

METHOD PUBLIC Clone : I_Datatype
VAR
    pClone : POINTER TO _TcVnVector2_USINT;
END_VAR
pClone := __NEW(_TcVnVector2_USINT);
Clone := pClone^;
END_METHOD

METHOD FB_init : BOOL
VAR_INPUT
	bInitRetains : BOOL; // if TRUE, the retain variables are initialized (warm start / cold start)
	bInCopyCode : BOOL;  // if TRUE, the instance afterwards gets moved into the copy code (online change)
	//InitialValue : <type>; // if possible, not all values can be initialized
END_VAR
//localData := InitialValue; // if possible, not all values can be initialized
SetBaseDatatypeReference();
AddBaseDatatype(aliasBaseDatatype);
END_METHOD

PROPERTY PUBLIC Identifier : T_MAXSTRING
GET
Identifier := 'TcVnVector2_USINT';
END_GET
END_PROPERTY

METHOD PUBLIC MakeReferenceTo
VAR_INPUT
	ReferenceTarget : REFERENCE TO TcVnVector2_USINT;
END_VAR
activeData REF= ReferenceTarget;
SetBaseDatatypeReference();
END_METHOD

METHOD PROTECTED SetBaseDatatypeReference
VAR_INPUT
END_VAR
aliasBaseDatatype.MakeReferenceTo(activeData);
END_METHOD

PROPERTY PUBLIC Size : UDINT
GET
Size := SIZEOF(activeData);
END_GET
END_PROPERTY

METHOD TryMakeReferenceTo : BOOL
VAR_INPUT
	Target : I_Datatype;
END_VAR
VAR
	pTargetData : POINTER TO TcVnVector2_USINT;
END_VAR
IF NOT IsEquivalentTo(Target) THEN
	RETURN;
END_IF

pTargetData := Target.Address;
activeData REF= pTargetData^;
SetBaseDatatypeReference();
TryMakeReferenceTo := TRUE;
END_METHOD

PROPERTY PUBLIC Value : REFERENCE TO TcVnVector2_USINT
GET
Value REF= activeData;
END_GET
END_PROPERTY

END_FUNCTION_BLOCK

// ---- Datatypes/Arrays/_Array0to1OfUSINT.TcPOU
{attribute 'linkalways'} 
{attribute 'no_explicit_call' := 'This FB is a CLASS and must be accessed using methods or properties'}
{attribute 'enable_dynamic_creation'}
FUNCTION_BLOCK _Array0to1OfUSINT EXTENDS ArrayDatatypeBase_1D
VAR CONSTANT
	lBound : DINT := 0;
	uBound : DINT := 1;
END_VAR
VAR
	localData : ARRAY [lBound..uBound] OF USINT;
	activeData : REFERENCE TO ARRAY [lBound..uBound] OF USINT REF= localData;
	elements : ARRAY [lBound..uBound] OF _USINT(0);
	baseType : _USINT(0);
END_VAR

PROPERTY PUBLIC Address : PVOID
GET
Address := ADR(activeData);
END_GET
END_PROPERTY

PROPERTY PUBLIC BaseDatatype : I_Datatype
GET
BaseDatatype := baseType;
END_GET
END_PROPERTY

METHOD PUBLIC ClearReference
VAR_INPUT
END_VAR
activeData REF= localData;
SetElementReference();
END_METHOD

METHOD PUBLIC Clone : I_Datatype
VAR
    pClone : POINTER TO _Array0to1OfUSINT;
END_VAR
pClone := __NEW(_Array0to1OfUSINT());
pClone^.Value := Value;
Clone := pClone^;
END_METHOD

METHOD FB_init : BOOL
VAR_INPUT
	bInitRetains : BOOL; // if TRUE, the retain variables are initialized (warm start / cold start)
	bInCopyCode : BOOL;  // if TRUE, the instance afterwards gets moved into the copy code (online change)
END_VAR
SetElementReference();
END_METHOD

METHOD PUBLIC MakeReferenceTo
VAR_INPUT
	ReferenceTarget : REFERENCE TO ARRAY [lBound..uBound] OF USINT;
END_VAR
activeData REF= ReferenceTarget;
SetElementReference();
END_METHOD

METHOD PROTECTED OnSerializeArrayValues
VAR_INPUT
	Serializer : I_Serializer;
END_VAR
VAR
	i : DINT;
END_VAR
FOR i := lBound TO uBound DO
	elements[i].SerializeWith(Serializer);
END_FOR
END_METHOD

METHOD PROTECTED SetElementReference
VAR_INPUT
END_VAR
VAR
	i : DINT;
END_VAR
FOR i := lBound TO uBound DO
	elements[i].MakeReferenceTo(activeData[i]);
END_FOR
END_METHOD

PROPERTY PUBLIC Size : UDINT
GET
Size := SIZEOF(activeData);
END_GET
END_PROPERTY

METHOD PROTECTED TryDeserializeArrayValues : BOOL
VAR_INPUT
	Deserializer : I_Deserializer;
	Feedback : I_DeserializerFeedback;
END_VAR
VAR
	enumerator : I_DeserializerArrayForwardEnumerator;
	i : DINT;
END_VAR
enumerator := Deserializer.GetArrayEnumerator();
i := lBound;

WHILE enumerator.MoveNext() AND i <= uBound DO
	
	IF NOT elements[i].TryDeserializeFrom(enumerator.Current, Feedback) THEN
		EXIT;
	END_IF
	i := i + 1;

END_WHILE
enumerator.Dispose();
END_METHOD

METHOD PUBLIC TryGetElementAsDatatypeByIndex : BOOL
VAR_INPUT
	Index : DINT;
	Destination : REFERENCE TO I_Datatype;
END_VAR
IF Index < lbound OR Index > ubound THEN
	RETURN;
END_IF

Destination := elements[Index];
TryGetElementAsDatatypeByIndex := TRUE;
END_METHOD

METHOD PUBLIC TryGetLowerBound : BOOL
VAR_INPUT
	Dimention : UDINT;
	Destination : REFERENCE TO DINT;
END_VAR
IF Dimention = 1 THEN
	Destination := lBound;
	TryGetLowerBound := TRUE;
END_IF
END_METHOD

METHOD PUBLIC TryGetUpperBound : BOOL
VAR_INPUT
	Dimention : UDINT;
	Destination : REFERENCE TO DINT;
END_VAR
IF Dimention = 1 THEN
	Destination := uBound;
	TryGetUpperBound := TRUE;
END_IF
END_METHOD

METHOD TryMakeReferenceTo : BOOL
VAR_INPUT
	Target : I_Datatype;
END_VAR
VAR
	pTargetData : POINTER TO ARRAY [lBound..uBound] OF USINT;
END_VAR
IF NOT IsEquivalentTo(Target) THEN
	RETURN;
END_IF

pTargetData := Target.Address;
activeData REF= pTargetData^;
SetElementReference();
TryMakeReferenceTo := TRUE;
END_METHOD

PROPERTY PUBLIC Value : REFERENCE TO ARRAY [lBound..uBound] OF USINT;
GET
Value ref= activeData;
END_GET
END_PROPERTY

END_FUNCTION_BLOCK

// ---- Datatypes/Aliases/_TcVnVector3_UINT.TcPOU
{attribute 'linkalways'} 
{attribute 'no_explicit_call' := 'This FB is a CLASS and must be accessed using methods or properties'}
{attribute 'enable_dynamic_creation'}
FUNCTION_BLOCK _TcVnVector3_UINT EXTENDS AliasDatatypeBase
VAR
	localData : TcVnVector3_UINT;
	activeData : REFERENCE TO TcVnVector3_UINT REF= localData;
	aliasBaseDatatype : _Array0to2OfUINT;
END_VAR

PROPERTY PUBLIC Address : PVOID
GET
Address := ADR(activeData);
END_GET
END_PROPERTY

METHOD PUBLIC ClearReference
VAR_INPUT
END_VAR
activeData REF= localData;
SetBaseDatatypeReference();
END_METHOD

METHOD PUBLIC Clone : I_Datatype
VAR
    pClone : POINTER TO _TcVnVector3_UINT;
END_VAR
pClone := __NEW(_TcVnVector3_UINT);
Clone := pClone^;
END_METHOD

METHOD FB_init : BOOL
VAR_INPUT
	bInitRetains : BOOL; // if TRUE, the retain variables are initialized (warm start / cold start)
	bInCopyCode : BOOL;  // if TRUE, the instance afterwards gets moved into the copy code (online change)
	//InitialValue : <type>; // if possible, not all values can be initialized
END_VAR
//localData := InitialValue; // if possible, not all values can be initialized
SetBaseDatatypeReference();
AddBaseDatatype(aliasBaseDatatype);
END_METHOD

PROPERTY PUBLIC Identifier : T_MAXSTRING
GET
Identifier := 'TcVnVector3_UINT';
END_GET
END_PROPERTY

METHOD PUBLIC MakeReferenceTo
VAR_INPUT
	ReferenceTarget : REFERENCE TO TcVnVector3_UINT;
END_VAR
activeData REF= ReferenceTarget;
SetBaseDatatypeReference();
END_METHOD

METHOD PROTECTED SetBaseDatatypeReference
VAR_INPUT
END_VAR
aliasBaseDatatype.MakeReferenceTo(activeData);
END_METHOD

PROPERTY PUBLIC Size : UDINT
GET
Size := SIZEOF(activeData);
END_GET
END_PROPERTY

METHOD TryMakeReferenceTo : BOOL
VAR_INPUT
	Target : I_Datatype;
END_VAR
VAR
	pTargetData : POINTER TO TcVnVector3_UINT;
END_VAR
IF NOT IsEquivalentTo(Target) THEN
	RETURN;
END_IF

pTargetData := Target.Address;
activeData REF= pTargetData^;
SetBaseDatatypeReference();
TryMakeReferenceTo := TRUE;
END_METHOD

PROPERTY PUBLIC Value : REFERENCE TO TcVnVector3_UINT
GET
Value REF= activeData;
END_GET
END_PROPERTY

END_FUNCTION_BLOCK

// ---- Datatypes/Aliases/_TcVnVector4_REAL.TcPOU
{attribute 'linkalways'} 
{attribute 'no_explicit_call' := 'This FB is a CLASS and must be accessed using methods or properties'}
{attribute 'enable_dynamic_creation'}
FUNCTION_BLOCK _TcVnVector4_REAL EXTENDS AliasDatatypeBase
VAR
	localData : TcVnVector4_REAL;
	activeData : REFERENCE TO TcVnVector4_REAL REF= localData;
	aliasBaseDatatype : _Array0to3OfREAL;
END_VAR

PROPERTY PUBLIC Address : PVOID
GET
Address := ADR(activeData);
END_GET
END_PROPERTY

METHOD PUBLIC ClearReference
VAR_INPUT
END_VAR
activeData REF= localData;
SetBaseDatatypeReference();
END_METHOD

METHOD PUBLIC Clone : I_Datatype
VAR
    pClone : POINTER TO _TcVnVector4_REAL;
END_VAR
pClone := __NEW(_TcVnVector4_REAL);
Clone := pClone^;
END_METHOD

METHOD FB_init : BOOL
VAR_INPUT
	bInitRetains : BOOL; // if TRUE, the retain variables are initialized (warm start / cold start)
	bInCopyCode : BOOL;  // if TRUE, the instance afterwards gets moved into the copy code (online change)
	//InitialValue : <type>; // if possible, not all values can be initialized
END_VAR
//localData := InitialValue; // if possible, not all values can be initialized
SetBaseDatatypeReference();
AddBaseDatatype(aliasBaseDatatype);
END_METHOD

PROPERTY PUBLIC Identifier : T_MAXSTRING
GET
Identifier := 'TcVnVector4_REAL';
END_GET
END_PROPERTY

METHOD PUBLIC MakeReferenceTo
VAR_INPUT
	ReferenceTarget : REFERENCE TO TcVnVector4_REAL;
END_VAR
activeData REF= ReferenceTarget;
SetBaseDatatypeReference();
END_METHOD

METHOD PROTECTED SetBaseDatatypeReference
VAR_INPUT
END_VAR
aliasBaseDatatype.MakeReferenceTo(activeData);
END_METHOD

PROPERTY PUBLIC Size : UDINT
GET
Size := SIZEOF(activeData);
END_GET
END_PROPERTY

METHOD TryMakeReferenceTo : BOOL
VAR_INPUT
	Target : I_Datatype;
END_VAR
VAR
	pTargetData : POINTER TO TcVnVector4_REAL;
END_VAR
IF NOT IsEquivalentTo(Target) THEN
	RETURN;
END_IF

pTargetData := Target.Address;
activeData REF= pTargetData^;
SetBaseDatatypeReference();
TryMakeReferenceTo := TRUE;
END_METHOD

PROPERTY PUBLIC Value : REFERENCE TO TcVnVector4_REAL
GET
Value REF= activeData;
END_GET
END_PROPERTY

END_FUNCTION_BLOCK

// ---- Datatypes/Arrays/_Array0to3OfREAL.TcPOU
{attribute 'linkalways'} 
{attribute 'no_explicit_call' := 'This FB is a CLASS and must be accessed using methods or properties'}
{attribute 'enable_dynamic_creation'}
FUNCTION_BLOCK _Array0to3OfREAL EXTENDS ArrayDatatypeBase_1D
VAR CONSTANT
	lBound : DINT := 0;
	uBound : DINT := 3;
END_VAR
VAR
	localData : ARRAY [lBound..uBound] OF REAL;
	activeData : REFERENCE TO ARRAY [lBound..uBound] OF REAL REF= localData;
	elements : ARRAY [lBound..uBound] OF _REAL(0.0);
	baseType : _REAL(0.0);
END_VAR

PROPERTY PUBLIC Address : PVOID
GET
Address := ADR(activeData);
END_GET
END_PROPERTY

PROPERTY PUBLIC BaseDatatype : I_Datatype
GET
BaseDatatype := baseType;
END_GET
END_PROPERTY

METHOD PUBLIC ClearReference
VAR_INPUT
END_VAR
activeData REF= localData;
SetElementReference();
END_METHOD

METHOD PUBLIC Clone : I_Datatype
VAR
    pClone : POINTER TO _Array0to3OfREAL;
END_VAR
pClone := __NEW(_Array0to3OfREAL());
pClone^.Value := Value;
Clone := pClone^;
END_METHOD

METHOD FB_init : BOOL
VAR_INPUT
	bInitRetains : BOOL; // if TRUE, the retain variables are initialized (warm start / cold start)
	bInCopyCode : BOOL;  // if TRUE, the instance afterwards gets moved into the copy code (online change)
END_VAR
SetElementReference();
END_METHOD

METHOD PUBLIC MakeReferenceTo
VAR_INPUT
	ReferenceTarget : REFERENCE TO ARRAY [lBound..uBound] OF REAL;
END_VAR
activeData REF= ReferenceTarget;
SetElementReference();
END_METHOD

METHOD PROTECTED OnSerializeArrayValues
VAR_INPUT
	Serializer : I_Serializer;
END_VAR
VAR
	i : DINT;
END_VAR
FOR i := lBound TO uBound DO
	elements[i].SerializeWith(Serializer);
END_FOR
END_METHOD

METHOD PROTECTED SetElementReference
VAR_INPUT
END_VAR
VAR
	i : DINT;
END_VAR
FOR i := lBound TO uBound DO
	elements[i].MakeReferenceTo(activeData[i]);
END_FOR
END_METHOD

PROPERTY PUBLIC Size : UDINT
GET
Size := SIZEOF(activeData);
END_GET
END_PROPERTY

METHOD PROTECTED TryDeserializeArrayValues : BOOL
VAR_INPUT
	Deserializer : I_Deserializer;
	Feedback : I_DeserializerFeedback;
END_VAR
VAR
	enumerator : I_DeserializerArrayForwardEnumerator;
	i : DINT;
END_VAR
enumerator := Deserializer.GetArrayEnumerator();
i := lBound;

WHILE enumerator.MoveNext() AND i <= uBound DO
	
	IF NOT elements[i].TryDeserializeFrom(enumerator.Current, Feedback) THEN
		EXIT;
	END_IF
	i := i + 1;

END_WHILE
enumerator.Dispose();
END_METHOD

